C01818=1070.032,30.785,434.123,172.808,24.822,154.487
C01819=1070.038,31.068,434.106,172.809,24.824,154.487
C01820=1070.044,31.317,434.090,172.810,24.827,154.487
C01821=1070.049,31.567,434.074,172.812,24.830,154.488
C01822=1070.056,31.816,434.059,172.813,24.833,154.488
C01823=1070.062,32.066,434.043,172.814,24.835,154.488
C01824=1070.068,32.315,434.027,172.816,24.838,154.489
C01825=1070.073,32.564,434.012,172.817,24.840,154.489
C01826=1070.079,32.814,433.996,172.818,24.843,154.489
C01827=1070.085,33.064,433.980,172.820,24.845,154.490
C01828=1070.091,33.313,433.964,172.821,24.848,154.490
C01829=1070.097,33.563,433.949,172.822,24.851,154.490
C01830=1070.103,33.812,433.933,172.824,24.854,154.491
C01831=1070.108,34.061,433.918,172.826,24.856,154.491
C01832=1070.115,34.310,433.902,172.827,24.859,154.491
C01833=1070.121,34.560,433.887,172.829,24.862,154.492
C01834=1070.127,34.810,433.870,172.830,24.865,154.492
C01835=1070.132,35.060,433.855,172.831,24.867,154.492
C01836=1070.139,35.309,433.839,172.832,24.870,154.493
C01837=1070.145,35.558,433.823,172.834,24.872,154.493
C01838=1070.150,35.807,433.808,172.835,24.875,154.493
C01839=1070.157,36.056,433.792,172.837,24.877,154.494
C01840=1070.162,36.306,433.777,172.838,24.880,154.494
C01841=1070.168,36.556,433.760,172.839,24.883,154.495
C01842=1070.174,36.805,433.744,172.841,24.885,154.495
C01843=1070.181,37.055,433.729,172.842,24.888,154.495
C01844=1070.187,37.304,433.713,172.843,24.890,154.495
C01845=1070.193,37.553,433.697,172.845,24.893,154.496
C01846=1070.198,37.803,433.681,172.846,24.896,154.496
C01847=1070.205,38.052,433.665,172.847,24.898,154.497
C01848=1070.210,38.301,433.649,172.849,24.901,154.497
C01849=1070.216,38.551,433.634,172.851,24.904,154.497
C01850=1070.222,38.800,433.618,172.852,24.906,154.497
C01851=1070.228,39.050,433.601,172.854,24.909,154.498
C01852=1070.233,39.300,433.586,172.855,24.912,154.498
C01853=1070.239,39.549,433.570,172.856,24.915,154.499
C01854=1070.245,39.798,433.553,172.858,24.917,154.499
C01855=1070.251,40.048,433.538,172.859,24.920,154.499
C01856=1070.256,40.297,433.522,172.860,24.923,154.500
C01857=1070.262,40.546,433.506,172.862,24.925,154.500
C01858=1070.268,40.796,433.489,172.863,24.928,154.500
C01859=1070.275,41.045,433.474,172.864,24.930,154.501
C01860=1070.281,41.295,433.458,172.866,24.933,154.501
C01861=1070.286,41.544,433.442,172.867,24.936,154.501
C01862=1070.292,41.793,433.426,172.868,24.939,154.502
C01863=1070.298,42.043,433.409,172.870,24.941,154.502
C01864=1070.304,42.293,433.394,172.871,24.944,154.502
C01865=1070.310,42.542,433.378,172.872,24.946,154.503
C01866=1070.316,42.791,433.361,172.875,24.949,154.503
C01867=1070.322,43.041,433.345,172.876,24.952,154.503
C01868=1070.328,43.290,433.329,172.877,24.955,154.504
C01869=1070.333,43.540,433.313,172.879,24.957,154.504
C01870=1070.339,43.789,433.297,172.880,24.960,154.504
C01871=1070.345,44.038,433.281,172.881,24.963,154.505
C01872=1070.351,44.287,433.265,172.883,24.965,154.505
C01873=1070.357,44.537,433.249,172.884,24.968,154.505
C01874=1070.363,44.786,433.232,172.885,24.970,154.506
C01875=1070.368,45.036,433.216,172.887,24.973,154.506
C01876=1070.374,45.285,433.199,172.888,24.976,154.507
C01877=1070.380,45.534,433.183,172.889,24.979,154.507
C01878=1070.385,45.784,433.168,172.891,24.981,154.507
C01879=1070.391,46.034,433.151,172.892,24.984,154.508
C01880=1070.398,46.316,433.132,172.894,24.988,154.508
C01881=1070.405,46.599,433.114,172.895,24.990,154.508
C01882=1070.411,46.882,433.096,172.897,24.993,154.509
C01883=1070.417,47.164,433.077,172.899,24.997,154.509
C01884=1070.423,47.413,433.061,172.900,25.000,154.510
C01885=1070.429,47.662,433.044,172.901,25.002,154.510
C01886=1070.435,47.912,433.028,172.903,25.005,154.510
C01887=1070.440,48.161,433.011,172.904,25.007,154.511
C01888=1070.446,48.411,432.995,172.905,25.010,154.511
C01889=1070.452,48.660,432.979,172.907,25.013,154.511
C01890=1070.458,48.909,432.963,172.908,25.015,154.512
C01891=1070.464,49.159,432.946,172.909,25.018,154.512
C01892=1070.469,49.408,432.929,172.911,25.021,154.512
C01893=1070.475,49.658,432.913,172.912,25.023,154.513
C01894=1070.481,49.907,432.897,172.913,25.026,154.513
C01895=1070.487,50.156,432.881,172.915,25.029,154.513
C01896=1070.493,50.406,432.864,172.917,25.032,154.514
C01897=1070.498,50.655,432.848,172.918,25.034,154.514
C01898=1070.504,50.905,432.831,172.920,25.037,154.514
C01899=1070.510,51.154,432.815,172.921,25.040,154.515
C01900=1070.517,51.404,432.798,172.922,25.042,154.515
C01901=1070.523,51.654,432.782,172.924,25.045,154.516
C01902=1070.528,51.903,432.765,172.925,25.048,154.516
C01903=1070.534,52.152,432.748,172.926,25.051,154.516
C01904=1070.540,52.401,432.732,172.928,25.053,154.517
C01905=1070.546,52.651,432.716,172.929,25.056,154.517
C01906=1070.551,52.900,432.699,172.930,25.059,154.517
C01907=1070.557,53.150,432.683,172.932,25.061,154.518
C01908=1070.563,53.399,432.666,172.933,25.064,154.518
C01909=1070.569,53.648,432.650,172.934,25.066,154.518
C01910=1070.575,53.897,432.633,172.937,25.069,154.519
C01911=1070.580,54.147,432.616,172.938,25.072,154.519
C01912=1070.586,54.396,432.600,172.939,25.075,154.519
C01913=1070.592,54.645,432.584,172.941,25.078,154.520
C01914=1070.598,54.896,432.567,172.942,25.080,154.520
C01915=1070.604,55.145,432.550,172.943,25.083,154.520
C01916=1070.610,55.394,432.533,172.945,25.085,154.521
C01917=1070.616,55.643,432.517,172.946,25.088,154.521
C01918=1070.622,55.893,432.500,172.948,25.090,154.521
C01919=1070.628,56.142,432.484,172.949,25.093,154.522
C01920=1070.634,56.391,432.467,172.950,25.096,154.522
C01921=1070.640,56.640,432.451,172.951,25.099,154.522
C01922=1070.646,56.891,432.434,172.953,25.101,154.523
C01923=1070.652,57.139,432.417,172.955,25.104,154.523
C01924=1070.658,57.389,432.400,172.956,25.107,154.524
C01925=1070.663,57.638,432.384,172.958,25.109,154.524
C01926=1070.669,57.888,432.367,172.959,25.112,154.524
C01927=1070.675,58.137,432.350,172.961,25.115,154.524
C01928=1070.682,58.387,432.334,172.962,25.117,154.525
C01929=1070.687,58.636,432.317,172.963,25.120,154.525
C01930=1070.693,58.885,432.300,172.965,25.123,154.526
C01931=1070.699,59.134,432.284,172.966,25.125,154.526
C01932=1070.704,59.384,432.267,172.967,25.128,154.526
C01933=1070.711,59.633,432.249,172.969,25.130,154.527
C01934=1070.717,59.883,432.233,172.970,25.133,154.527
C01935=1070.722,60.132,432.216,172.971,25.136,154.527
C01936=1070.729,60.381,432.199,172.974,25.139,154.528
C01937=1070.735,60.630,432.183,172.975,25.141,154.528
C01938=1070.741,60.880,432.165,172.976,25.144,154.528
C01939=1070.747,61.130,432.149,172.978,25.146,154.529
C01940=1070.753,61.379,432.133,172.979,25.149,154.529
C01941=1070.758,61.628,432.115,172.980,25.152,154.529
C01942=1070.765,61.878,432.098,172.982,25.154,154.530
C01943=1070.771,62.127,432.081,172.983,25.157,154.530
C01944=1070.777,62.410,432.063,172.985,25.160,154.530
C01945=1070.784,62.691,432.043,172.987,25.163,154.531
C01946=1070.791,62.974,432.024,172.988,25.166,154.531
C01947=1070.798,63.256,432.005,172.990,25.169,154.531
C01948=1070.803,63.506,431.989,172.992,25.172,154.532
C01949=1070.810,63.755,431.971,172.993,25.174,154.532
C01950=1070.816,64.005,431.955,172.994,25.177,154.532
C01951=1070.821,64.254,431.937,172.996,25.179,154.533
C01952=1070.828,64.504,431.921,172.997,25.182,154.533
C01953=1070.834,64.753,431.903,172.998,25.185,154.534
C01954=1070.839,65.002,431.887,173.000,25.188,154.534
C01955=1070.845,65.251,431.869,173.001,25.190,154.534
C01956=1070.851,65.502,431.852,173.002,25.193,154.535
C01957=1070.857,65.750,431.835,173.005,25.195,154.535
C01958=1070.863,65.999,431.818,173.006,25.198,154.535
C01959=1070.869,66.249,431.801,173.007,25.201,154.536
C01960=1070.875,66.498,431.783,173.009,25.204,154.536
C01961=1070.881,66.748,431.767,173.010,25.206,154.536
C01962=1070.886,66.997,431.750,173.012,25.209,154.537
C01963=1070.892,67.246,431.732,173.013,25.212,154.537
C01964=1070.898,67.496,431.715,173.014,25.214,154.537
C01965=1070.904,67.745,431.698,173.016,25.217,154.538
C01966=1070.910,67.994,431.682,173.017,25.220,154.538
C01967=1070.915,68.243,431.664,173.019,25.222,154.538
C01968=1070.921,68.493,431.646,173.020,25.225,154.539
C01969=1070.927,68.742,431.630,173.022,25.228,154.539
C01970=1070.933,68.991,431.612,173.023,25.230,154.539
C01971=1070.939,69.241,431.594,173.025,25.233,154.540
C01972=1070.945,69.491,431.578,173.026,25.236,154.540
C01973=1070.950,69.740,431.560,173.027,25.239,154.541
C01974=1070.957,69.988,431.543,173.029,25.241,154.541
C01975=1070.962,70.239,431.526,173.030,25.244,154.541
C01976=1070.968,70.488,431.509,173.031,25.246,154.542
C01977=1070.973,70.737,431.491,173.034,25.249,154.542
C01978=1070.980,70.986,431.474,173.035,25.252,154.542
C01979=1070.986,71.236,431.457,173.036,25.255,154.543
C01980=1070.991,71.485,431.439,173.038,25.257,154.543
C01981=1070.997,71.735,431.421,173.039,25.260,154.543
C01982=1071.003,71.983,431.404,173.040,25.263,154.544
C01983=1071.009,72.233,431.388,173.042,25.265,154.544
C01984=1071.015,72.483,431.370,173.043,25.268,154.544
C01985=1071.020,72.732,431.352,173.044,25.271,154.545
C01986=1071.027,72.981,431.335,173.046,25.273,154.545
C01987=1071.032,73.230,431.318,173.048,25.276,154.545
C01988=1071.038,73.480,431.300,173.050,25.279,154.546
C01989=1071.043,73.729,431.283,173.051,25.281,154.546
C01990=1071.049,73.978,431.265,173.052,25.284,154.547
C01991=1071.056,74.227,431.248,173.054,25.287,154.547
C01992=1071.061,74.476,431.230,173.055,25.290,154.547
C01993=1071.067,74.726,431.212,173.056,25.292,154.548
C01994=1071.073,74.976,431.196,173.058,25.295,154.548
C01995=1071.078,75.225,431.178,173.059,25.298,154.548
C01996=1071.085,75.474,431.161,173.061,25.300,154.549
C01997=1071.091,75.723,431.143,173.063,25.303,154.549
C01998=1071.096,75.972,431.126,173.064,25.306,154.549
C01999=1071.102,76.222,431.108,173.065,25.308,154.550
C02000=1071.108,76.471,431.090,173.067,25.311,154.550
C02001=1071.115,76.721,431.073,173.068,25.314,154.550
C02002=1071.120,76.970,431.055,173.070,25.316,154.551
C02003=1071.126,77.219,431.038,173.071,25.319,154.551
C02004=1071.131,77.469,431.020,173.072,25.322,154.551
C02005=1071.137,77.718,431.003,173.075,25.324,154.552
C02006=1071.143,77.968,430.985,173.076,25.327,154.552
C02007=1071.149,78.217,430.967,173.077,25.330,154.552
C02008=1071.155,78.499,430.947,173.079,25.332,154.553
C02009=1071.162,78.781,430.927,173.081,25.336,154.553
C02010=1071.169,79.064,430.907,173.082,25.338,154.554
C02011=1071.176,79.346,430.887,173.083,25.342,154.554
C02012=1071.181,79.595,430.870,173.086,25.345,154.554
C02013=1071.187,79.845,430.852,173.087,25.347,154.555
C02014=1071.193,80.094,430.834,173.088,25.350,154.555
C02015=1071.197,80.343,430.816,173.090,25.353,154.555
C02016=1071.204,80.593,430.798,173.091,25.356,154.556
C02017=1071.209,80.842,430.781,173.092,25.358,154.556
C02018=1071.215,81.092,430.763,173.094,25.361,154.557
C02019=1071.221,81.341,430.745,173.095,25.364,154.557
C02020=1071.227,81.590,430.727,173.097,25.366,154.557
C02021=1071.233,81.839,430.709,173.099,25.369,154.558
C02022=1071.238,82.088,430.691,173.100,25.371,154.558
C02023=1071.244,82.338,430.673,173.102,25.374,154.558
C02024=1071.250,82.587,430.656,173.103,25.377,154.559
C02025=1071.256,82.836,430.638,173.104,25.380,154.559
C02026=1071.261,83.085,430.620,173.106,25.382,154.559
C02027=1071.268,83.335,430.602,173.107,25.385,154.560
C02028=1071.273,83.584,430.584,173.109,25.388,154.560
C02029=1071.280,83.833,430.566,173.111,25.391,154.560
C02030=1071.285,84.082,430.549,173.112,25.393,154.561
C02031=1071.291,84.331,430.531,173.113,25.396,154.561
C02032=1071.296,84.581,430.513,173.115,25.398,154.561
C02033=1071.301,84.830,430.495,173.116,25.401,154.562
C02034=1071.308,85.080,430.476,173.117,25.404,154.562
C02035=1071.313,85.329,430.459,173.120,25.407,154.562
C02036=1071.320,85.578,430.441,173.121,25.410,154.563
C02037=1071.325,85.827,430.423,173.123,25.412,154.563
C02038=1071.331,86.077,430.405,173.124,25.415,154.564
C02039=1071.337,86.326,430.387,173.125,25.417,154.564
C02040=1071.343,86.575,430.369,173.127,25.420,154.564
C02041=1071.349,86.825,430.351,173.128,25.423,154.565
C02042=1071.355,87.073,430.333,173.129,25.425,154.565
C02043=1071.360,87.324,430.314,173.132,25.428,154.565
C02044=1071.366,87.573,430.297,173.133,25.431,154.566
C02045=1071.372,87.822,430.279,173.134,25.433,154.566
C02046=1071.378,88.071,430.261,173.136,25.436,154.566
C02047=1071.384,88.320,430.243,173.137,25.439,154.567
C02048=1071.390,88.570,430.225,173.139,25.441,154.567
C02049=1071.396,88.819,430.207,173.141,25.444,154.567
C02050=1071.402,89.068,430.189,173.142,25.447,154.568
C02051=1071.407,89.318,430.170,173.144,25.449,154.568
C02052=1071.413,89.567,430.152,173.145,25.452,154.568
C02053=1071.419,89.816,430.134,173.146,25.455,154.569
C02054=1071.425,90.066,430.116,173.148,25.457,154.569
C02055=1071.431,90.314,430.098,173.149,25.460,154.569
C02056=1071.437,90.564,430.080,173.152,25.462,154.570
C02057=1071.443,90.813,430.061,173.153,25.465,154.570
C02058=1071.448,91.062,430.043,173.154,25.468,154.570
C02059=1071.454,91.312,430.025,173.156,25.470,154.571
C02060=1071.460,91.560,430.007,173.157,25.473,154.571
C02061=1071.465,91.810,429.988,173.158,25.476,154.571
C02062=1071.471,92.059,429.970,173.160,25.478,154.572
C02063=1071.477,92.309,429.952,173.162,25.482,154.572
C02064=1071.482,92.557,429.933,173.163,25.484,154.573
C02065=1071.489,92.807,429.915,173.165,25.487,154.573
C02066=1071.494,93.057,429.897,173.166,25.489,154.573
C02067=1071.500,93.306,429.879,173.167,25.492,154.574
C02068=1071.506,93.555,429.861,173.169,25.495,154.574
C02069=1071.511,93.804,429.842,173.171,25.498,154.574
C02070=1071.517,94.054,429.824,173.173,25.500,154.575
C02071=1071.524,94.303,429.805,173.174,25.503,154.575
C02072=1071.530,94.585,429.784,173.175,25.506,154.575
C02073=1071.536,94.868,429.764,173.178,25.509,154.576
C02074=1071.542,95.150,429.743,173.179,25.512,154.576
C02075=1071.550,95.432,429.722,173.181,25.515,154.577
C02076=1071.555,95.681,429.703,173.182,25.518,154.577
C02077=1071.561,95.931,429.685,173.184,25.521,154.577
C02078=1071.566,96.180,429.666,173.185,25.523,154.578
C02079=1071.572,96.429,429.648,173.187,25.526,154.578
C02080=1071.578,96.678,429.630,173.189,25.528,154.578
C02081=1071.583,96.928,429.611,173.190,25.531,154.579
C02082=1071.590,97.177,429.593,173.192,25.534,154.579
C02083=1071.595,97.426,429.574,173.193,25.536,154.579
C02084=1071.601,97.675,429.556,173.194,25.539,154.580
C02085=1071.607,97.924,429.537,173.196,25.542,154.580
C02086=1071.613,98.174,429.518,173.198,25.545,154.580
C02087=1071.618,98.423,429.501,173.200,25.547,154.581
C02088=1071.624,98.672,429.481,173.201,25.550,154.581
C02089=1071.631,98.921,429.463,173.202,25.552,154.581
C02090=1071.636,99.172,429.444,173.204,25.555,154.582
C02091=1071.642,99.420,429.426,173.205,25.557,154.582
C02092=1071.648,99.669,429.407,173.207,25.561,154.582
C02093=1071.654,99.919,429.389,173.209,25.563,154.583
C02094=1071.659,100.168,429.370,173.210,25.566,154.583
C02095=1071.665,100.417,429.351,173.212,25.568,154.583
C02096=1071.671,100.666,429.332,173.213,25.571,154.584
C02097=1071.677,100.916,429.314,173.215,25.574,154.584
C02098=1071.683,101.165,429.296,173.217,25.576,154.585
C02099=1071.688,101.414,429.276,173.218,25.579,154.585
C02100=1071.695,101.663,429.258,173.219,25.582,154.585
C02101=1071.700,101.912,429.240,173.221,25.584,154.586
C02102=1071.705,102.162,429.220,173.223,25.587,154.586
C02103=1071.712,102.411,429.202,173.224,25.590,154.586
C02104=1071.717,102.660,429.183,173.226,25.592,154.587
C02105=1071.722,102.909,429.164,173.227,25.595,154.587
C02106=1071.729,103.159,429.146,173.229,25.597,154.587
C02107=1071.734,103.408,429.127,173.230,25.600,154.588
C02108=1071.739,103.657,429.108,173.232,25.603,154.588
C02109=1071.746,103.906,429.089,173.234,25.606,154.588
C02110=1071.751,104.156,429.070,173.235,25.609,154.589
C02111=1071.757,104.404,429.051,173.237,25.611,154.589
C02112=1071.763,104.654,429.033,173.238,25.614,154.589
C02113=1071.768,104.904,429.014,173.240,25.616,154.590
C02114=1071.774,105.153,428.994,173.242,25.619,154.590
C02115=1071.780,105.401,428.976,173.243,25.622,154.590
C02116=1071.786,105.651,428.957,173.244,25.624,154.591
C02117=1071.791,105.900,428.938,173.246,25.627,154.591
C02118=1071.798,106.149,428.919,173.248,25.630,154.591
C02119=1071.803,106.398,428.900,173.249,25.633,154.592
C02120=1071.808,106.648,428.881,173.251,25.635,154.592
C02121=1071.815,106.897,428.862,173.252,25.638,154.593
C02122=1071.821,107.146,428.843,173.254,25.640,154.593
C02123=1071.826,107.396,428.824,173.256,25.643,154.593
C02124=1071.832,107.644,428.805,173.257,25.646,154.593
C02125=1071.838,107.893,428.786,173.259,25.648,154.594
C02126=1071.843,108.143,428.767,173.260,25.651,154.594
C02127=1071.849,108.392,428.748,173.263,25.654,154.595
C02128=1071.856,108.641,428.729,173.264,25.656,154.595
C02129=1071.861,108.890,428.710,173.265,25.659,154.595
C02130=1071.866,109.140,428.691,173.267,25.661,154.596
C02131=1071.873,109.389,428.672,173.268,25.664,154.596
C02132=1071.878,109.638,428.653,173.271,25.667,154.596
C02133=1071.884,109.888,428.634,173.272,25.670,154.597
C02134=1071.890,110.137,428.615,173.273,25.672,154.597
C02135=1071.896,110.385,428.596,173.275,25.675,154.597
C02136=1071.902,110.668,428.574,173.277,25.678,154.598
C02137=1071.909,110.950,428.552,173.278,25.681,154.598
C02138=1071.915,111.233,428.531,173.281,25.684,154.598
C02139=1071.922,111.516,428.509,173.282,25.687,154.599
C02140=1071.928,111.765,428.490,173.284,25.690,154.599
C02141=1071.933,112.014,428.471,173.286,25.692,154.599
C02142=1071.939,112.263,428.451,173.287,25.695,154.600
C02143=1071.944,112.512,428.432,173.288,25.698,154.600
C02144=1071.951,112.761,428.413,173.290,25.700,154.600
C02145=1071.957,113.011,428.394,173.292,25.703,154.601
C02146=1071.962,113.260,428.375,173.294,25.705,154.601
C02147=1071.968,113.509,428.356,173.295,25.708,154.602
C02148=1071.974,113.758,428.336,173.296,25.710,154.602
C02149=1071.980,114.008,428.317,173.299,25.714,154.602
C02150=1071.985,114.256,428.298,173.300,25.716,154.602
C02151=1071.990,114.506,428.278,173.302,25.719,154.603
C02152=1071.996,114.755,428.259,173.303,25.722,154.603
C02153=1072.002,115.004,428.239,173.305,25.724,154.604
C02154=1072.008,115.254,428.220,173.307,25.727,154.604
C02155=1072.013,115.503,428.201,173.308,25.729,154.604
C02156=1072.019,115.751,428.181,173.309,25.732,154.605
C02157=1072.025,116.000,428.162,173.312,25.735,154.605
C02158=1072.030,116.250,428.143,173.313,25.738,154.605
C02159=1072.036,116.499,428.123,173.314,25.741,154.606
C02160=1072.042,116.748,428.103,173.316,25.743,154.606
C02161=1072.047,116.998,428.084,173.317,25.746,154.606
C02162=1072.053,117.247,428.064,173.320,25.749,154.607
C02163=1072.058,117.495,428.045,173.321,25.751,154.607
C02164=1072.064,117.745,428.026,173.322,25.754,154.608
C02165=1072.069,117.994,428.006,173.324,25.756,154.608
C02166=1072.075,118.243,427.986,173.326,25.759,154.608
C02167=1072.081,118.493,427.967,173.328,25.762,154.608
C02168=1072.087,118.742,427.948,173.329,25.765,154.609
C02169=1072.093,118.991,427.928,173.330,25.767,154.609
C02170=1072.098,119.240,427.909,173.333,25.770,154.610
C02171=1072.104,119.489,427.888,173.334,25.773,154.610
C02172=1072.109,119.739,427.869,173.336,25.775,154.610
C02173=1072.115,119.988,427.850,173.338,25.778,154.611
C02174=1072.121,120.237,427.830,173.339,25.781,154.611
C02175=1072.126,120.486,427.811,173.341,25.783,154.611
C02176=1072.132,120.735,427.791,173.342,25.786,154.612
C02177=1072.138,120.984,427.772,173.344,25.789,154.612
C02178=1072.143,121.233,427.751,173.346,25.791,154.612
C02179=1072.149,121.483,427.732,173.347,25.794,154.613
C02180=1072.155,121.731,427.712,173.349,25.796,154.613
C02181=1072.160,121.981,427.693,173.351,25.799,154.613
C02182=1072.166,122.230,427.673,173.352,25.802,154.614
C02183=1072.172,122.479,427.653,173.354,25.805,154.614
C02184=1072.178,122.728,427.633,173.355,25.807,154.614
C02185=1072.183,122.978,427.614,173.358,25.810,154.615
C02186=1072.189,123.226,427.594,173.359,25.812,154.615
C02187=1072.195,123.476,427.574,173.360,25.815,154.615
C02188=1072.201,123.725,427.554,173.363,25.818,154.616
C02189=1072.206,123.974,427.535,173.364,25.821,154.616
C02190=1072.212,124.223,427.515,173.366,25.823,154.616
C02191=1072.217,124.473,427.495,173.367,25.826,154.617
C02192=1072.223,124.721,427.475,173.369,25.828,154.617
C02193=1072.229,124.970,427.455,173.371,25.831,154.617
C02194=1072.235,125.220,427.436,173.372,25.833,154.618
C02195=1072.241,125.469,427.416,173.374,25.837,154.618
C02196=1072.246,125.718,427.396,173.376,25.839,154.618
C02197=1072.253,125.968,427.376,173.377,25.842,154.619
C02198=1072.259,126.217,427.356,173.379,25.844,154.619
C02199=1072.264,126.466,427.337,173.381,25.847,154.619
C02200=1072.270,126.748,427.314,173.382,25.850,154.620
C02201=1072.277,127.031,427.292,173.385,25.853,154.620
C02202=1072.284,127.313,427.269,173.387,25.856,154.620
C02203=1072.290,127.595,427.247,173.388,25.859,154.621
C02204=1072.296,127.844,427.227,173.390,25.861,154.621
C02205=1072.301,128.093,427.206,173.392,25.864,154.621
C02206=1072.308,128.343,427.187,173.394,25.866,154.622
C02207=1072.314,128.592,427.167,173.395,25.869,154.622
C02208=1072.319,128.841,427.147,173.397,25.872,154.622
C02209=1072.325,129.090,427.126,173.399,25.875,154.623
C02210=1072.330,129.339,427.107,173.400,25.877,154.623
C02211=1072.336,129.588,427.087,173.403,25.880,154.624
C02212=1072.342,129.837,427.067,173.404,25.882,154.624
C02213=1072.348,130.086,427.046,173.406,25.885,154.624
C02214=1072.354,130.336,427.027,173.407,25.887,154.625
C02215=1072.360,130.585,427.007,173.409,25.890,154.625
C02216=1072.366,130.834,426.987,173.411,25.893,154.625
C02217=1072.371,131.083,426.966,173.412,25.895,154.625
C02218=1072.377,131.332,426.946,173.415,25.898,154.626
C02219=1072.383,131.580,426.926,173.416,25.901,154.626
C02220=1072.389,131.831,426.907,173.417,25.903,154.626
C02221=1072.395,132.080,426.886,173.420,25.906,154.627
C02222=1072.401,132.329,426.866,173.421,25.908,154.627
C02223=1072.406,132.578,426.846,173.423,25.911,154.627
C02224=1072.412,132.827,426.826,173.425,25.914,154.628
C02225=1072.417,133.076,426.805,173.426,25.917,154.628
C02226=1072.423,133.324,426.785,173.428,25.919,154.628
C02227=1072.429,133.574,426.764,173.430,25.922,154.629
C02228=1072.435,133.823,426.744,173.432,25.924,154.629
C02229=1072.440,134.073,426.725,173.433,25.927,154.629
C02230=1072.446,134.322,426.705,173.435,25.930,154.630
C02231=1072.451,134.571,426.684,173.437,25.932,154.630
C02232=1072.457,134.820,426.664,173.438,25.935,154.630
C02233=1072.463,135.069,426.644,173.441,25.937,154.631
C02234=1072.469,135.318,426.623,173.442,25.940,154.631
C02235=1072.474,135.567,426.603,173.443,25.943,154.631
C02236=1072.480,135.816,426.583,173.446,25.946,154.632
C02237=1072.486,136.065,426.562,173.447,25.948,154.632
C02238=1072.492,136.314,426.542,173.449,25.951,154.632
C02239=1072.497,136.564,426.521,173.451,25.953,154.633
C02240=1072.503,136.813,426.501,173.452,25.956,154.633
C02241=1072.509,137.062,426.481,173.454,25.959,154.633
C02242=1072.514,137.311,426.460,173.456,25.962,154.634
C02243=1072.520,137.560,426.440,173.458,25.964,154.634
C02244=1072.526,137.809,426.419,173.459,25.966,154.634
C02245=1072.532,138.058,426.399,173.461,25.969,154.635
C02246=1072.537,138.307,426.378,173.463,25.972,154.635
C02247=1072.543,138.556,426.358,173.464,25.974,154.635
C02248=1072.549,138.805,426.338,173.467,25.977,154.636
C02249=1072.555,139.055,426.317,173.468,25.980,154.636
C02250=1072.561,139.304,426.297,173.471,25.982,154.636
C02251=1072.566,139.553,426.276,173.472,25.985,154.637
C02252=1072.571,139.802,426.256,173.473,25.988,154.637
C02253=1072.578,140.051,426.235,173.476,25.990,154.637
C02254=1072.583,140.300,426.214,173.477,25.993,154.638
C02255=1072.589,140.549,426.194,173.479,25.995,154.638
C02256=1072.594,140.798,426.174,173.481,25.998,154.638
C02257=1072.600,141.048,426.153,173.482,26.001,154.639
C02258=1072.606,141.296,426.131,173.484,26.004,154.639
C02259=1072.612,141.545,426.111,173.486,26.006,154.639
C02260=1072.617,141.794,426.091,173.488,26.009,154.640
C02261=1072.623,142.044,426.070,173.490,26.012,154.640
C02262=1072.628,142.293,426.049,173.491,26.014,154.640
C02263=1072.635,142.541,426.029,173.493,26.017,154.641
C02264=1072.640,142.824,426.005,173.495,26.020,154.641
C02265=1072.647,143.106,425.982,173.497,26.023,154.641
C02266=1072.654,143.388,425.958,173.499,26.026,154.642
C02267=1072.659,143.670,425.935,173.501,26.029,154.642
C02268=1072.665,143.920,425.913,173.503,26.032,154.643
C02269=1072.671,144.168,425.893,173.505,26.034,154.643
C02270=1072.677,144.418,425.873,173.506,26.037,154.643
C02271=1072.683,144.667,425.851,173.509,26.040,154.644
C02272=1072.688,144.916,425.831,173.510,26.042,154.644
C02273=1072.694,145.165,425.811,173.512,26.045,154.644
C02274=1072.700,145.414,425.789,173.514,26.047,154.645
C02275=1072.706,145.663,425.769,173.515,26.050,154.645
C02276=1072.711,145.912,425.747,173.518,26.053,154.645
C02277=1072.717,146.161,425.726,173.519,26.056,154.646
C02278=1072.723,146.410,425.706,173.521,26.058,154.646
C02279=1072.728,146.659,425.685,173.523,26.060,154.646
C02280=1072.734,146.909,425.664,173.524,26.063,154.647
C02281=1072.740,147.157,425.643,173.527,26.066,154.647
C02282=1072.745,147.406,425.622,173.528,26.069,154.647
C02283=1072.751,147.656,425.601,173.530,26.071,154.648
C02284=1072.757,147.904,425.581,173.532,26.074,154.648
C02285=1072.763,148.154,425.560,173.534,26.076,154.648
C02286=1072.769,148.403,425.539,173.536,26.079,154.648
C02287=1072.774,148.652,425.518,173.537,26.082,154.649
C02288=1072.780,148.901,425.496,173.540,26.084,154.649
C02289=1072.785,149.150,425.476,173.541,26.087,154.650
C02290=1072.791,149.398,425.455,173.543,26.089,154.650
C02291=1072.797,149.648,425.434,173.545,26.093,154.650
C02292=1072.802,149.897,425.412,173.546,26.095,154.651
C02293=1072.808,150.146,425.392,173.549,26.098,154.651
C02294=1072.814,150.395,425.370,173.550,26.100,154.651
C02295=1072.819,150.644,425.349,173.552,26.103,154.652
C02296=1072.825,150.893,425.328,173.554,26.106,154.652
C02297=1072.831,151.142,425.307,173.555,26.108,154.652
C02298=1072.836,151.391,425.286,173.558,26.111,154.653
C02299=1072.842,151.640,425.265,173.559,26.114,154.653
C02300=1072.847,151.889,425.244,173.562,26.116,154.653
C02301=1072.854,152.139,425.222,173.563,26.119,154.653
C02302=1072.859,152.387,425.201,173.565,26.121,154.654
C02303=1072.864,152.636,425.181,173.567,26.124,154.654
C02304=1072.871,152.885,425.159,173.568,26.127,154.655
C02305=1072.876,153.134,425.138,173.571,26.129,154.655
C02306=1072.882,153.384,425.117,173.572,26.132,154.655
C02307=1072.888,153.632,425.095,173.575,26.135,154.655
C02308=1072.894,153.882,425.074,173.576,26.138,154.656
C02309=1072.899,154.131,425.053,173.578,26.140,154.656
C02310=1072.904,154.380,425.031,173.580,26.143,154.657
C02311=1072.910,154.629,425.010,173.581,26.145,154.657
C02312=1072.916,154.877,424.988,173.584,26.148,154.657
C02313=1072.921,155.127,424.968,173.585,26.151,154.658
C02314=1072.927,155.375,424.946,173.588,26.153,154.658
C02315=1072.933,155.625,424.925,173.589,26.156,154.658
C02316=1072.939,155.873,424.903,173.591,26.159,154.658
C02317=1072.945,156.123,424.882,173.593,26.161,154.659
C02318=1072.949,156.372,424.861,173.595,26.164,154.659
C02319=1072.956,156.621,424.839,173.597,26.167,154.660
C02320=1072.961,156.870,424.818,173.599,26.169,154.660
C02321=1072.967,157.119,424.796,173.600,26.172,154.660
C02322=1072.973,157.368,424.776,173.603,26.175,154.660
C02323=1072.978,157.617,424.753,173.604,26.178,154.661
C02324=1072.984,157.866,424.732,173.606,26.180,154.661
C02325=1072.990,158.115,424.710,173.608,26.182,154.661
C02326=1072.995,158.364,424.689,173.610,26.185,154.662
C02327=1073.001,158.613,424.667,173.612,26.188,154.662
C02328=1073.007,158.895,424.643,173.614,26.191,154.662
C02329=1073.014,159.177,424.618,173.617,26.194,154.663
C02330=1073.020,159.459,424.594,173.618,26.197,154.663
C02331=1073.027,159.741,424.570,173.620,26.200,154.664
C02332=1073.032,159.989,424.548,173.623,26.203,154.664
C02333=1073.038,160.239,424.526,173.624,26.205,154.664
C02334=1073.044,160.487,424.505,173.627,26.208,154.665
C02335=1073.050,160.737,424.484,173.628,26.211,154.665
C02336=1073.054,160.986,424.462,173.630,26.213,154.665
C02337=1073.061,161.235,424.441,173.632,26.216,154.666
C02338=1073.067,161.484,424.419,173.634,26.219,154.666
C02339=1073.072,161.733,424.397,173.636,26.221,154.666
C02340=1073.078,161.982,424.376,173.638,26.224,154.667
C02341=1073.083,162.231,424.354,173.639,26.227,154.667
C02342=1073.089,162.480,424.331,173.642,26.229,154.667
C02343=1073.094,162.728,424.310,173.643,26.232,154.668
C02344=1073.100,162.978,424.288,173.646,26.235,154.668
C02345=1073.105,163.226,424.266,173.647,26.238,154.668
C02346=1073.110,163.476,424.244,173.649,26.241,154.669
C02347=1073.116,163.725,424.223,173.651,26.243,154.669
C02348=1073.121,163.974,424.200,173.653,26.246,154.669
C02349=1073.127,164.223,424.179,173.655,26.249,154.670
C02350=1073.132,164.472,424.157,173.657,26.251,154.670
C02351=1073.138,164.721,424.136,173.659,26.254,154.670
C02352=1073.143,164.970,424.113,173.661,26.257,154.671
C02353=1073.149,165.218,424.091,173.662,26.260,154.671
C02354=1073.155,165.467,424.069,173.665,26.263,154.672
C02355=1073.159,165.716,424.047,173.666,26.265,154.672
C02356=1073.166,165.965,424.026,173.668,26.268,154.672
C02357=1073.171,166.215,424.003,173.670,26.270,154.672
C02358=1073.177,166.463,423.981,173.672,26.273,154.673
C02359=1073.182,166.712,423.959,173.674,26.276,154.673
C02360=1073.187,166.961,423.937,173.676,26.279,154.674
C02361=1073.193,167.210,423.916,173.678,26.281,154.674
C02362=1073.199,167.460,423.893,173.680,26.284,154.674
C02363=1073.205,167.708,423.871,173.681,26.287,154.675
C02364=1073.210,167.957,423.849,173.684,26.290,154.675
C02365=1073.215,168.206,423.827,173.686,26.293,154.675
C02366=1073.221,168.455,423.805,173.688,26.295,154.676
C02367=1073.227,168.704,423.783,173.690,26.298,154.676
C02368=1073.232,168.953,423.762,173.692,26.300,154.676
C02369=1073.238,169.202,423.739,173.694,26.303,154.677
C02370=1073.243,169.451,423.716,173.695,26.306,154.677
C02371=1073.249,169.700,423.695,173.698,26.309,154.677
C02372=1073.254,169.949,423.673,173.699,26.311,154.678
C02373=1073.260,170.198,423.650,173.702,26.314,154.678
C02374=1073.266,170.447,423.629,173.704,26.317,154.678
C02375=1073.271,170.696,423.606,173.705,26.319,154.679
C02376=1073.278,170.945,423.584,173.708,26.322,154.679
C02377=1073.282,171.194,423.562,173.709,26.325,154.679
C02378=1073.288,171.442,423.539,173.712,26.328,154.680
C02379=1073.294,171.692,423.518,173.713,26.330,154.680
C02380=1073.299,171.940,423.496,173.715,26.333,154.680
C02381=1073.305,172.189,423.473,173.717,26.336,154.681
C02382=1073.311,172.439,423.451,173.719,26.339,154.681
C02383=1073.317,172.687,423.428,173.722,26.341,154.681
C02384=1073.322,172.936,423.406,173.723,26.344,154.682
C02385=1073.328,173.185,423.384,173.726,26.347,154.682
C02386=1073.333,173.434,423.362,173.727,26.349,154.682
C02387=1073.339,173.683,423.339,173.729,26.352,154.683
C02388=1073.345,173.932,423.318,173.732,26.355,154.683
C02389=1073.350,174.181,423.295,173.733,26.357,154.683
C02390=1073.356,174.430,423.272,173.736,26.360,154.684
C02391=1073.362,174.679,423.249,173.737,26.363,154.684
C02392=1073.368,174.960,423.225,173.739,26.366,154.684
C02393=1073.375,175.242,423.199,173.742,26.369,154.685
C02394=1073.381,175.523,423.174,173.744,26.372,154.685
C02395=1073.388,175.805,423.149,173.746,26.375,154.686
C02396=1073.393,176.054,423.126,173.749,26.378,154.686
C02397=1073.399,176.302,423.104,173.750,26.380,154.686
C02398=1073.404,176.552,423.081,173.753,26.383,154.686
C02399=1073.410,176.801,423.059,173.755,26.386,154.687
C02400=1073.416,177.050,423.037,173.757,26.388,154.687
C02401=1073.422,177.299,423.014,173.759,26.391,154.687
C02402=1073.428,177.548,422.992,173.760,26.394,154.688
C02403=1073.433,177.796,422.970,173.763,26.396,154.688
C02404=1073.439,178.045,422.947,173.765,26.399,154.688
C02405=1073.444,178.294,422.924,173.767,26.401,154.689
C02406=1073.451,178.543,422.902,173.769,26.405,154.689
C02407=1073.456,178.792,422.879,173.771,26.407,154.689
C02408=1073.462,179.041,422.856,173.773,26.410,154.690
C02409=1073.467,179.291,422.834,173.775,26.412,154.690
C02410=1073.474,179.539,422.812,173.777,26.415,154.690
C02411=1073.479,179.787,422.789,173.779,26.418,154.691
C02412=1073.485,180.036,422.766,173.782,26.420,154.691
C02413=1073.490,180.286,422.744,173.783,26.423,154.691
C02414=1073.496,180.535,422.721,173.786,26.426,154.692
C02415=1073.502,180.783,422.699,173.788,26.429,154.692
C02416=1073.508,181.032,422.676,173.789,26.431,154.692
C02417=1073.514,181.281,422.653,173.792,26.434,154.693
C02418=1073.519,181.531,422.630,173.794,26.437,154.693
C02419=1073.526,181.779,422.608,173.796,26.439,154.693
C02420=1073.531,182.028,422.585,173.798,26.442,154.694
C02421=1073.537,182.277,422.562,173.800,26.444,154.694
C02422=1073.543,182.526,422.539,173.802,26.447,154.694
C02423=1073.549,182.775,422.516,173.804,26.450,154.695
C02424=1073.554,183.024,422.493,173.806,26.452,154.695
C02425=1073.561,183.273,422.472,173.808,26.455,154.695
C02426=1073.566,183.522,422.449,173.811,26.458,154.696
C02427=1073.572,183.771,422.426,173.812,26.461,154.696
C02428=1073.578,184.020,422.403,173.815,26.463,154.696
C02429=1073.583,184.269,422.380,173.817,26.466,154.697
C02430=1073.590,184.517,422.358,173.819,26.468,154.697
C02431=1073.596,184.766,422.335,173.821,26.471,154.697
C02432=1073.601,185.015,422.312,173.823,26.474,154.698
C02433=1073.606,185.263,422.289,173.826,26.477,154.698
C02434=1073.612,185.512,422.266,173.827,26.479,154.698
C02435=1073.617,185.761,422.243,173.830,26.482,154.699
C02436=1073.623,186.010,422.220,173.832,26.486,154.699
C02437=1073.628,186.259,422.196,173.833,26.488,154.699
C02438=1073.634,186.508,422.173,173.836,26.491,154.700
C02439=1073.639,186.757,422.150,173.838,26.494,154.700
C02440=1073.645,187.006,422.127,173.840,26.496,154.700
C02441=1073.650,187.255,422.104,173.842,26.499,154.701
C02442=1073.656,187.504,422.081,173.844,26.502,154.701
C02443=1073.661,187.752,422.058,173.846,26.505,154.701
C02444=1073.667,188.001,422.035,173.848,26.508,154.702
C02445=1073.672,188.250,422.011,173.851,26.511,154.702
C02446=1073.678,188.499,421.988,173.852,26.513,154.702
C02447=1073.683,188.748,421.965,173.854,26.516,154.703
C02448=1073.689,188.996,421.942,173.857,26.519,154.703
C02449=1073.694,189.246,421.919,173.859,26.522,154.703
C02450=1073.700,189.495,421.896,173.861,26.524,154.704
C02451=1073.706,189.743,421.872,173.863,26.527,154.704
C02452=1073.712,189.992,421.849,173.865,26.530,154.705
C02453=1073.717,190.241,421.826,173.867,26.533,154.705
C02454=1073.722,190.490,421.803,173.869,26.535,154.705
C02455=1073.728,190.739,421.780,173.872,26.539,154.706
C02456=1073.735,191.020,421.753,173.874,26.542,154.706
C02457=1073.740,191.301,421.727,173.876,26.545,154.706
C02458=1073.747,191.583,421.700,173.879,26.548,154.707
C02459=1073.754,191.864,421.674,173.881,26.551,154.707
C02460=1073.759,192.113,421.650,173.883,26.554,154.708
C02461=1073.765,192.362,421.627,173.886,26.557,154.708
C02462=1073.771,192.610,421.604,173.887,26.559,154.708
C02463=1073.776,192.859,421.580,173.890,26.562,154.709
C02464=1073.782,193.108,421.557,173.892,26.565,154.709
C02465=1073.788,193.356,421.533,173.895,26.568,154.709
C02466=1073.793,193.606,421.510,173.896,26.571,154.710
C02467=1073.798,193.854,421.487,173.898,26.574,154.710
C02468=1073.804,194.103,421.463,173.901,26.576,154.710
C02469=1073.809,194.352,421.440,173.903,26.579,154.711
C02470=1073.815,194.601,421.417,173.905,26.582,154.711
C02471=1073.821,194.849,421.393,173.907,26.585,154.711
C02472=1073.827,195.099,421.369,173.909,26.588,154.712
C02473=1073.833,195.347,421.346,173.912,26.590,154.712
C02474=1073.838,195.596,421.322,173.913,26.593,154.712
C02475=1073.844,195.845,421.298,173.916,26.596,154.713
C02476=1073.850,196.094,421.275,173.918,26.599,154.713
C02477=1073.855,196.343,421.252,173.920,26.602,154.713
C02478=1073.861,196.591,421.228,173.922,26.604,154.714
C02479=1073.866,196.840,421.205,173.924,26.607,154.714
C02480=1073.872,197.089,421.181,173.927,26.610,154.715
C02481=1073.878,197.338,421.158,173.929,26.613,154.715
C02482=1073.883,197.587,421.133,173.932,26.616,154.715
C02483=1073.889,197.835,421.110,173.933,26.618,154.715
C02484=1073.895,198.084,421.087,173.935,26.621,154.716
C02485=1073.901,198.333,421.062,173.938,26.624,154.716
C02486=1073.907,198.582,421.039,173.940,26.627,154.717
C02487=1073.912,198.831,421.015,173.942,26.629,154.717
C02488=1073.918,199.080,420.992,173.944,26.632,154.717
C02489=1073.924,199.328,420.968,173.947,26.635,154.718
C02490=1073.930,199.577,420.944,173.949,26.638,154.718
C02491=1073.935,199.826,420.921,173.951,26.641,154.718
C02492=1073.941,200.075,420.897,173.954,26.644,154.719
C02493=1073.946,200.324,420.874,173.955,26.646,154.719
C02494=1073.952,200.573,420.849,173.958,26.649,154.719
C02495=1073.958,200.821,420.825,173.960,26.652,154.720
C02496=1073.964,201.070,420.802,173.962,26.655,154.720
C02497=1073.969,201.319,420.778,173.965,26.658,154.720
C02498=1073.976,201.568,420.754,173.966,26.660,154.721
C02499=1073.981,201.816,420.730,173.969,26.663,154.721
C02500=1073.987,202.065,420.707,173.971,26.666,154.721
C02501=1073.992,202.314,420.683,173.974,26.668,154.722
C02502=1073.999,202.563,420.659,173.976,26.672,154.722
C02503=1074.004,202.811,420.634,173.978,26.675,154.722
C02504=1074.009,203.060,420.611,173.980,26.677,154.723
C02505=1074.015,203.309,420.587,173.982,26.680,154.723
C02506=1074.021,203.558,420.563,173.985,26.683,154.724
C02507=1074.026,203.807,420.538,173.987,26.686,154.724
C02508=1074.032,204.055,420.514,173.989,26.689,154.724
C02509=1074.038,204.304,420.491,173.992,26.692,154.725
C02510=1074.043,204.553,420.467,173.993,26.694,154.725
C02511=1074.049,204.802,420.442,173.996,26.697,154.725
C02512=1074.055,205.050,420.419,173.998,26.701,154.726
C02513=1074.060,205.299,420.394,174.000,26.703,154.726
C02514=1074.066,205.548,420.370,174.003,26.706,154.726
C02515=1074.071,205.797,420.345,174.005,26.709,154.727
C02516=1074.077,206.045,420.322,174.007,26.712,154.727
C02517=1074.083,206.295,420.298,174.009,26.715,154.728
C02518=1074.088,206.544,420.274,174.011,26.718,154.728
C02519=1074.094,206.792,420.250,174.014,26.721,154.728
C02520=1074.118,207.831,420.148,174.137,26.785,154.729
C02521=1074.127,208.246,420.107,174.140,26.791,154.730
C02522=1074.137,208.660,420.065,174.144,26.798,154.731
C02523=1074.147,209.075,420.025,174.147,26.804,154.732
C02524=1074.156,209.489,419.982,174.150,26.811,154.733
C02525=1074.162,209.738,419.958,174.153,26.814,154.733
C02526=1074.168,209.986,419.933,174.155,26.818,154.734
C02527=1074.174,210.235,419.907,174.157,26.822,154.735
C02528=1074.180,210.484,419.883,174.159,26.826,154.735
C02529=1074.185,210.732,419.858,174.161,26.830,154.736
C02530=1074.191,210.981,419.833,174.164,26.834,154.736
C02531=1074.197,211.230,419.808,174.165,26.837,154.737
C02532=1074.203,211.478,419.783,174.167,26.841,154.738
C02533=1074.208,211.728,419.758,174.169,26.845,154.738
C02534=1074.214,211.976,419.732,174.172,26.849,154.739
C02535=1074.220,212.224,419.707,174.174,26.852,154.739
C02536=1074.226,212.474,419.683,174.176,26.856,154.740
C02537=1074.232,212.722,419.657,174.178,26.860,154.740
C02538=1074.238,212.970,419.632,174.180,26.864,154.741
C02539=1074.243,213.220,419.607,174.183,26.868,154.741
C02540=1074.249,213.469,419.582,174.185,26.872,154.742
C02541=1074.255,213.717,419.557,174.186,26.875,154.743
C02542=1074.261,213.965,419.532,174.188,26.879,154.743
C02543=1074.266,214.215,419.506,174.191,26.883,154.744
C02544=1074.272,214.463,419.481,174.193,26.887,154.744
C02545=1074.278,214.711,419.456,174.195,26.891,154.745
C02546=1074.283,214.960,419.430,174.197,26.895,154.746
C02547=1074.289,215.208,419.405,174.200,26.898,154.746
C02548=1074.295,215.458,419.381,174.202,26.902,154.747
C02549=1074.300,215.707,419.355,174.204,26.906,154.747
C02550=1074.306,215.955,419.330,174.206,26.910,154.748
C02551=1074.312,216.203,419.304,174.208,26.914,154.749
C02552=1074.318,216.452,419.279,174.211,26.918,154.749
C02553=1074.324,216.701,419.253,174.212,26.921,154.750
C02554=1074.329,216.949,419.228,174.214,26.925,154.750
C02555=1074.336,217.198,419.203,174.217,26.929,154.751
C02556=1074.341,217.447,419.178,174.219,26.933,154.751
C02557=1074.347,217.696,419.152,174.221,26.936,154.752
C02558=1074.352,217.944,419.127,174.223,26.940,154.753
C02559=1074.358,218.193,419.101,174.225,26.944,154.753
C02560=1074.364,218.441,419.076,174.228,26.948,154.754
C02561=1074.370,218.690,419.050,174.230,26.952,154.754
C02562=1074.376,218.939,419.025,174.232,26.956,154.755
C02563=1074.382,219.187,419.000,174.234,26.959,154.755
C02564=1074.387,219.436,418.974,174.237,26.963,154.756
C02565=1074.393,219.685,418.948,174.239,26.967,154.757
C02566=1074.399,219.933,418.923,174.241,26.971,154.757
C02567=1074.405,220.182,418.897,174.243,26.975,154.758
C02568=1074.411,220.430,418.871,174.246,26.978,154.758
C02569=1074.416,220.679,418.846,174.247,26.982,154.759
C02570=1074.423,220.927,418.820,174.249,26.986,154.759
C02571=1074.429,221.176,418.795,174.251,26.990,154.760
C02572=1074.434,221.425,418.769,174.254,26.993,154.761
C02573=1074.444,221.844,418.726,174.257,27.000,154.762
C02574=1074.454,222.262,418.683,174.261,27.006,154.762
C02575=1074.464,222.681,418.639,174.265,27.013,154.764
C02576=1074.473,223.100,418.596,174.269,27.019,154.764
C02577=1074.479,223.349,418.570,174.271,27.023,154.765
C02578=1074.485,223.598,418.544,174.273,27.027,154.766
C02579=1074.490,223.845,418.518,174.275,27.030,154.766
C02580=1074.496,224.094,418.492,174.278,27.034,154.767
C02581=1074.502,224.343,418.467,174.280,27.038,154.767
C02582=1074.507,224.592,418.441,174.282,27.042,154.768
C02583=1074.513,224.840,418.414,174.284,27.046,154.768
C02584=1074.519,225.089,418.389,174.286,27.050,154.769
C02585=1074.525,225.338,418.363,174.289,27.053,154.770
C02586=1074.531,225.586,418.337,174.291,27.057,154.770
C02587=1074.537,225.835,418.311,174.293,27.061,154.771
C02588=1074.542,226.083,418.285,174.295,27.065,154.771
C02589=1074.548,226.331,418.259,174.298,27.069,154.772
C02590=1074.554,226.580,418.233,174.300,27.073,154.773
C02591=1074.559,226.829,418.208,174.302,27.076,154.773
C02592=1074.565,227.077,418.182,174.305,27.080,154.774
C02593=1074.571,227.326,418.156,174.307,27.084,154.774
C02594=1074.577,227.575,418.129,174.309,27.087,154.775
C02595=1074.583,227.823,418.104,174.311,27.091,154.775
C02596=1074.589,228.072,418.077,174.314,27.095,154.776
C02597=1074.594,228.321,418.051,174.316,27.099,154.776
C02598=1074.601,228.569,418.025,174.318,27.103,154.777
C02599=1074.606,228.818,417.999,174.320,27.106,154.778
C02600=1074.612,229.066,417.972,174.323,27.110,154.778
C02601=1074.617,229.315,417.946,174.325,27.114,154.779
C02602=1074.624,229.563,417.920,174.327,27.117,154.779
C02603=1074.629,229.812,417.894,174.329,27.121,154.780
C02604=1074.635,230.060,417.868,174.332,27.125,154.780
C02605=1074.641,230.309,417.842,174.334,27.129,154.781
C02606=1074.647,230.557,417.816,174.336,27.133,154.782
C02607=1074.653,230.806,417.790,174.338,27.137,154.782
C02608=1074.658,231.055,417.763,174.341,27.140,154.783
C02609=1074.664,231.303,417.737,174.343,27.144,154.783
C02610=1074.670,231.552,417.711,174.345,27.148,154.784
C02611=1074.675,231.800,417.684,174.347,27.152,154.785
C02612=1074.681,232.049,417.657,174.350,27.156,154.785
C02613=1074.687,232.298,417.631,174.352,27.159,154.786
C02614=1074.692,232.546,417.605,174.354,27.163,154.786
C02615=1074.700,232.795,417.578,174.357,27.167,154.787
C02616=1074.705,233.044,417.552,174.359,27.171,154.787
C02617=1074.711,233.292,417.526,174.361,27.174,154.788
C02618=1074.717,233.541,417.499,174.363,27.178,154.789
C02619=1074.722,233.789,417.472,174.366,27.182,154.789
C02620=1074.728,234.038,417.447,174.368,27.186,154.790
C02621=1074.734,234.286,417.420,174.371,27.190,154.790
C02622=1074.739,234.535,417.393,174.373,27.194,154.791
C02623=1074.745,234.783,417.367,174.376,27.198,154.791
C02624=1074.751,235.031,417.340,174.378,27.202,154.792
C02625=1074.760,235.442,417.296,174.382,27.208,154.793
C02626=1074.769,235.853,417.252,174.385,27.214,154.794
C02627=1074.779,236.263,417.208,174.389,27.220,154.795
C02628=1074.789,236.673,417.164,174.393,27.227,154.796
C02629=1074.795,236.922,417.138,174.395,27.230,154.796
C02630=1074.800,237.170,417.111,174.398,27.234,154.797
C02631=1074.806,237.419,417.084,174.400,27.238,154.798
C02632=1074.812,237.667,417.058,174.402,27.241,154.798
C02633=1074.818,237.916,417.031,174.404,27.245,154.799
C02634=1074.824,238.164,417.004,174.407,27.249,154.799
C02635=1074.830,238.413,416.977,174.409,27.253,154.800
C02636=1074.835,238.661,416.950,174.411,27.256,154.800
C02637=1074.841,238.910,416.923,174.414,27.261,154.801
C02638=1074.847,239.159,416.896,174.417,27.264,154.802
C02639=1074.853,239.407,416.870,174.419,27.268,154.802
C02640=1074.859,239.655,416.843,174.421,27.272,154.803
C02641=1074.864,239.904,416.816,174.424,27.276,154.803
C02642=1074.870,240.152,416.790,174.426,27.280,154.804
C02643=1074.877,240.401,416.763,174.428,27.283,154.804
C02644=1074.882,240.650,416.736,174.430,27.287,154.805
C02645=1074.887,240.898,416.709,174.433,27.291,154.806
C02646=1074.893,241.147,416.682,174.435,27.294,154.806
C02647=1074.899,241.395,416.656,174.437,27.298,154.807
C02648=1074.906,241.643,416.628,174.440,27.302,154.807
C02649=1074.911,241.892,416.601,174.442,27.306,154.808
C02650=1074.916,242.140,416.574,174.445,27.310,154.808
C02651=1074.923,242.390,416.547,174.448,27.313,154.809
C02652=1074.928,242.638,416.520,174.450,27.317,154.810
C02653=1074.935,242.886,416.493,174.452,27.321,154.810
C02654=1074.940,243.134,416.466,174.454,27.325,154.811
C02655=1074.946,243.383,416.439,174.457,27.328,154.811
C02656=1074.952,243.632,416.412,174.459,27.332,154.812
C02657=1074.957,243.880,416.384,174.461,27.336,154.812
C02658=1074.963,244.128,416.357,174.463,27.340,154.813
C02659=1074.969,244.377,416.330,174.467,27.344,154.814
C02660=1074.975,244.625,416.302,174.469,27.348,154.814
C02661=1074.980,244.874,416.276,174.471,27.351,154.815
C02662=1074.985,245.122,416.249,174.474,27.355,154.815
C02663=1074.992,245.371,416.221,174.476,27.359,154.816
C02664=1074.998,245.619,416.194,174.478,27.363,154.817
C02665=1075.003,245.868,416.167,174.480,27.367,154.817
C02666=1075.010,246.116,416.139,174.483,27.371,154.818
C02667=1075.015,246.365,416.112,174.486,27.374,154.818
C02668=1075.021,246.613,416.085,174.488,27.378,154.819
C02669=1075.027,246.862,416.058,174.491,27.382,154.819
C02670=1075.032,247.110,416.030,174.493,27.386,154.820
C02671=1075.037,247.358,416.002,174.495,27.390,154.821
C02672=1075.043,247.607,415.976,174.497,27.394,154.821
C02673=1075.049,247.856,415.947,174.500,27.397,154.822
C02674=1075.055,248.104,415.921,174.502,27.401,154.822
C02675=1075.060,248.352,415.893,174.505,27.405,154.823
C02676=1075.066,248.601,415.864,174.507,27.409,154.823
C02677=1075.075,249.004,415.820,174.511,27.415,154.824
C02678=1075.085,249.408,415.776,174.515,27.421,154.825
C02679=1075.094,249.812,415.731,174.519,27.428,154.826
C02680=1075.103,250.215,415.686,174.523,27.434,154.827
C02681=1075.109,250.465,415.659,174.525,27.438,154.828
C02682=1075.115,250.713,415.631,174.527,27.441,154.828
C02683=1075.120,250.961,415.603,174.531,27.446,154.829
C02684=1075.127,251.210,415.576,174.533,27.449,154.830
C02685=1075.132,251.458,415.548,174.535,27.453,154.830
C02686=1075.137,251.706,415.520,174.538,27.457,154.831
C02687=1075.144,251.955,415.493,174.540,27.461,154.831
C02688=1075.149,252.203,415.465,174.542,27.464,154.832
C02689=1075.155,252.452,415.436,174.545,27.469,154.833
C02690=1075.161,252.699,415.409,174.548,27.472,154.833
C02691=1075.167,252.949,415.382,174.550,27.476,154.834
C02692=1075.172,253.197,415.354,174.552,27.480,154.834
C02693=1075.178,253.445,415.326,174.555,27.484,154.835
C02694=1075.184,253.693,415.298,174.557,27.487,154.835
C02695=1075.189,253.941,415.270,174.560,27.492,154.836
C02696=1075.196,254.190,415.242,174.562,27.495,154.837
C02697=1075.201,254.438,415.215,174.565,27.499,154.837
C02698=1075.207,254.687,415.187,174.567,27.503,154.838
C02699=1075.212,254.935,415.159,174.569,27.507,154.838
C02700=1075.219,255.184,415.131,174.573,27.511,154.839
C02701=1075.224,255.432,415.103,174.575,27.515,154.840
C02702=1075.230,255.681,415.075,174.577,27.518,154.840
C02703=1075.236,255.929,415.047,174.580,27.522,154.841
C02704=1075.242,256.177,415.019,174.582,27.526,154.841
C02705=1075.248,256.425,414.991,174.585,27.530,154.842
C02706=1075.254,256.674,414.963,174.587,27.533,154.842
C02707=1075.260,256.922,414.935,174.590,27.537,154.843
C02708=1075.266,257.170,414.907,174.592,27.541,154.844
C02709=1075.272,257.419,414.879,174.594,27.544,154.844
C02710=1075.277,257.667,414.851,174.598,27.549,154.845
C02711=1075.283,257.916,414.822,174.600,27.552,154.845
C02712=1075.289,258.164,414.795,174.602,27.556,154.846
C02713=1075.295,258.412,414.767,174.605,27.560,154.846
C02714=1075.301,258.661,414.738,174.608,27.564,154.847
C02715=1075.306,258.909,414.710,174.610,27.568,154.848
C02716=1075.313,259.158,414.683,174.612,27.572,154.848
C02717=1075.318,259.406,414.655,174.615,27.575,154.849
C02718=1075.324,259.654,414.626,174.617,27.579,154.849
C02719=1075.330,259.903,414.598,174.620,27.583,154.850
C02720=1075.336,260.151,414.569,174.623,27.586,154.850
C02721=1075.342,260.399,414.542,174.625,27.590,154.851
C02722=1075.348,260.648,414.513,174.627,27.594,154.852
C02723=1075.354,260.896,414.485,174.631,27.598,154.852
C02724=1075.360,261.145,414.457,174.633,27.602,154.853
C02725=1075.366,261.393,414.428,174.635,27.606,154.853
C02726=1075.372,261.640,414.401,174.638,27.609,154.854
C02727=1075.378,261.889,414.372,174.641,27.613,154.854
C02728=1075.384,262.138,414.344,174.643,27.617,154.855
C02729=1075.393,262.539,414.298,174.647,27.623,154.856
C02730=1075.403,262.940,414.252,174.651,27.629,154.857
C02731=1075.413,263.341,414.207,174.656,27.635,154.858
C02732=1075.422,263.742,414.161,174.660,27.641,154.859
C02733=1075.428,263.990,414.132,174.662,27.645,154.859
C02734=1075.434,264.239,414.104,174.664,27.649,154.860
C02735=1075.440,264.487,414.075,174.668,27.653,154.860
C02736=1075.445,264.736,414.046,174.670,27.657,154.861
C02737=1075.452,264.984,414.017,174.672,27.661,154.862
C02738=1075.457,265.233,413.989,174.675,27.664,154.862
C02739=1075.463,265.481,413.961,174.678,27.669,154.863
C02740=1075.469,265.729,413.932,174.680,27.672,154.863
C02741=1075.475,265.978,413.903,174.683,27.676,154.864
C02742=1075.481,266.225,413.875,174.685,27.680,154.865
C02743=1075.486,266.474,413.846,174.688,27.684,154.865
C02744=1075.492,266.722,413.817,174.690,27.688,154.866
C02745=1075.498,266.970,413.788,174.693,27.691,154.866
C02746=1075.504,267.218,413.760,174.696,27.696,154.867
C02747=1075.510,267.466,413.731,174.698,27.699,154.868
C02748=1075.516,267.715,413.702,174.701,27.703,154.868
C02749=1075.521,267.964,413.673,174.703,27.707,154.869
C02750=1075.527,268.211,413.644,174.706,27.711,154.869
C02751=1075.533,268.460,413.616,174.709,27.715,154.870
C02752=1075.539,268.708,413.587,174.711,27.718,154.871
C02753=1075.545,268.957,413.558,174.714,27.723,154.871
C02754=1075.551,269.205,413.529,174.717,27.726,154.872
C02755=1075.556,269.453,413.500,174.719,27.730,154.872
C02756=1075.563,269.701,413.471,174.722,27.734,154.873
C02757=1075.569,269.949,413.443,174.724,27.738,154.874
C02758=1075.574,270.198,413.413,174.727,27.742,154.874
C02759=1075.580,270.446,413.384,174.729,27.745,154.875
C02760=1075.586,270.693,413.355,174.732,27.750,154.875
C02761=1075.591,270.943,413.326,174.735,27.754,154.876
C02762=1075.597,271.191,413.297,174.737,27.757,154.876
C02763=1075.604,271.439,413.268,174.740,27.761,154.877
C02764=1075.609,271.687,413.239,174.743,27.765,154.878
C02765=1075.615,271.935,413.210,174.745,27.769,154.878
C02766=1075.621,272.183,413.182,174.748,27.773,154.879
C02767=1075.626,272.432,413.152,174.751,27.777,154.879
C02768=1075.632,272.680,413.123,174.753,27.781,154.880
C02769=1075.639,272.928,413.094,174.756,27.785,154.881
C02770=1075.644,273.177,413.064,174.759,27.788,154.881
C02771=1075.650,273.425,413.035,174.761,27.792,154.882
C02772=1075.656,273.673,413.006,174.764,27.796,154.882
C02773=1075.662,273.921,412.977,174.766,27.800,154.883
C02774=1075.667,274.169,412.947,174.769,27.804,154.884
C02775=1075.673,274.417,412.918,174.772,27.808,154.884
C02776=1075.680,274.665,412.889,174.774,27.812,154.885
C02777=1075.685,274.914,412.860,174.777,27.816,154.886
C02778=1075.691,275.162,412.831,174.780,27.820,154.886
C02779=1075.697,275.410,412.801,174.782,27.824,154.887
C02780=1075.703,275.658,412.772,174.785,27.828,154.887
C02781=1075.712,276.063,412.724,174.790,27.834,154.888
C02782=1075.722,276.467,412.676,174.793,27.840,154.889
C02783=1075.731,276.872,412.628,174.798,27.847,154.890
C02784=1075.741,277.276,412.580,174.802,27.853,154.891
C02785=1075.746,277.524,412.550,174.804,27.857,154.892
C02786=1075.753,277.772,412.521,174.808,27.861,154.892
C02787=1075.758,278.021,412.492,174.810,27.865,154.893
C02788=1075.765,278.268,412.462,174.813,27.869,154.894
C02789=1075.770,278.517,412.432,174.816,27.873,154.894
C02790=1075.776,278.765,412.403,174.818,27.877,154.895
C02791=1075.782,279.013,412.374,174.821,27.881,154.896
C02792=1075.788,279.261,412.343,174.824,27.885,154.896
C02793=1075.794,279.509,412.314,174.826,27.888,154.897
C02794=1075.799,279.758,412.285,174.829,27.893,154.897
C02795=1075.805,280.006,412.255,174.832,27.897,154.898
C02796=1075.812,280.254,412.225,174.835,27.901,154.899
C02797=1075.817,280.502,412.196,174.837,27.904,154.899
C02798=1075.823,280.751,412.166,174.840,27.908,154.900
C02799=1075.829,280.998,412.136,174.843,27.912,154.900
C02800=1075.835,281.246,412.107,174.845,27.916,154.901
C02801=1075.840,281.494,412.076,174.848,27.920,154.902
C02802=1075.846,281.743,412.047,174.851,27.924,154.902
C02803=1075.851,281.991,412.017,174.853,27.928,154.903
C02804=1075.858,282.239,411.987,174.856,27.932,154.904
C02805=1075.864,282.487,411.958,174.859,27.936,154.904
C02806=1075.869,282.735,411.927,174.861,27.940,154.905
C02807=1075.875,282.983,411.898,174.864,27.944,154.905
C02808=1075.881,283.231,411.867,174.867,27.948,154.906
C02809=1075.887,283.479,411.838,174.870,27.952,154.907
C02810=1075.893,283.727,411.808,174.872,27.956,154.907
C02811=1075.899,283.976,411.778,174.875,27.960,154.908
C02812=1075.905,284.224,411.748,174.878,27.964,154.908
C02813=1075.910,284.472,411.717,174.880,27.968,154.909
C02814=1075.916,284.720,411.688,174.884,27.972,154.910
C02815=1075.922,284.968,411.657,174.886,27.976,154.910
C02816=1075.928,285.216,411.628,174.889,27.980,154.911
C02817=1075.934,285.464,411.598,174.891,27.984,154.912
C02818=1075.940,285.712,411.567,174.894,27.988,154.912
C02819=1075.945,285.960,411.538,174.897,27.992,154.913
C02820=1075.952,286.209,411.507,174.899,27.996,154.914
C02821=1075.957,286.457,411.477,174.903,28.000,154.914
C02822=1075.963,286.705,411.447,174.905,28.004,154.915
C02823=1075.969,286.953,411.417,174.908,28.009,154.915
C02824=1075.975,287.201,411.386,174.911,28.012,154.916
C02825=1075.981,287.448,411.357,174.913,28.016,154.917
C02826=1075.987,287.698,411.327,174.916,28.020,154.917
C02827=1075.993,287.945,411.296,174.919,28.024,154.918
C02828=1075.999,288.193,411.266,174.922,28.028,154.919
C02829=1076.005,288.441,411.236,174.924,28.032,154.919
C02830=1076.011,288.690,411.205,174.928,28.036,154.920
C02831=1076.017,288.938,411.175,174.930,28.040,154.920
C02832=1076.022,289.186,411.145,174.933,28.044,154.921
C02833=1076.032,289.599,411.094,174.937,28.051,154.922
C02834=1076.042,290.015,411.043,174.942,28.058,154.923
C02835=1076.052,290.429,410.993,174.947,28.065,154.924
C02836=1076.062,290.843,410.941,174.952,28.071,154.925
C02837=1076.068,291.091,410.911,174.954,28.075,154.926
C02838=1076.074,291.339,410.881,174.957,28.080,154.927
C02839=1076.080,291.586,410.850,174.960,28.084,154.927
C02840=1076.085,291.835,410.819,174.963,28.088,154.928
C02841=1076.091,292.083,410.789,174.965,28.092,154.929
C02842=1076.097,292.331,410.758,174.969,28.096,154.929
C02843=1076.103,292.579,410.728,174.971,28.100,154.930
C02844=1076.109,292.827,410.697,174.974,28.104,154.930
C02845=1076.115,293.075,410.667,174.977,28.108,154.931
C02846=1076.120,293.323,410.636,174.980,28.112,154.932
C02847=1076.127,293.572,410.605,174.982,28.116,154.932
C02848=1076.133,293.819,410.574,174.985,28.121,154.933
C02849=1076.138,294.067,410.544,174.988,28.125,154.934
C02850=1076.145,294.315,410.513,174.991,28.129,154.934
C02851=1076.150,294.563,410.482,174.993,28.133,154.935
C02852=1076.156,294.811,410.452,174.997,28.137,154.936
C02853=1076.162,295.059,410.420,174.999,28.141,154.936
C02854=1076.168,295.307,410.390,175.002,28.145,154.937
C02855=1076.173,295.555,410.359,175.005,28.149,154.938
C02856=1076.180,295.804,410.328,175.008,28.153,154.938
C02857=1076.186,296.051,410.297,175.010,28.157,154.939
C02858=1076.192,296.299,410.267,175.014,28.161,154.940
C02859=1076.197,296.548,410.236,175.016,28.165,154.940
C02860=1076.204,296.795,410.204,175.019,28.170,154.941
C02861=1076.209,297.043,410.174,175.022,28.174,154.941
C02862=1076.215,297.291,410.143,175.025,28.178,154.942
C02863=1076.221,297.539,410.112,175.027,28.182,154.943
C02864=1076.227,297.787,410.080,175.031,28.186,154.943
C02865=1076.233,298.035,410.050,175.033,28.190,154.944
C02866=1076.238,298.283,410.018,175.036,28.195,154.945
C02867=1076.244,298.531,409.988,175.039,28.199,154.945
C02868=1076.250,298.779,409.956,175.042,28.203,154.946
C02869=1076.256,299.027,409.926,175.044,28.207,154.947
C02870=1076.262,299.275,409.894,175.047,28.211,154.948
C02871=1076.267,299.523,409.863,175.051,28.216,154.948
C02872=1076.273,299.770,409.832,175.053,28.220,154.949
C02873=1076.279,300.019,409.800,175.056,28.224,154.950
C02874=1076.285,300.266,409.769,175.059,28.228,154.950
C02875=1076.291,300.514,409.737,175.062,28.232,154.951
C02876=1076.296,300.762,409.707,175.064,28.237,154.952
C02877=1076.302,301.010,409.675,175.068,28.241,154.952
C02878=1076.308,301.259,409.644,175.070,28.245,154.953
C02879=1076.314,301.506,409.613,175.073,28.249,154.954
C02880=1076.320,301.754,409.581,175.076,28.254,154.954
C02881=1076.325,302.002,409.550,175.079,28.258,154.955
C02882=1076.331,302.250,409.518,175.082,28.262,154.956
C02883=1076.337,302.498,409.487,175.084,28.267,154.956
C02884=1076.343,302.746,409.456,175.088,28.271,154.957
C02885=1076.347,302.960,409.428,175.090,28.274,154.958
C02886=1076.353,303.175,409.401,175.093,28.278,154.958
C02887=1076.358,303.388,409.374,175.095,28.281,154.959
C02888=1076.363,303.603,409.347,175.097,28.285,154.960
C02889=1076.368,303.818,409.319,175.100,28.289,154.960
C02890=1076.373,304.032,409.293,175.102,28.293,154.961
C02891=1076.379,304.246,409.265,175.106,28.296,154.961
C02892=1076.383,304.462,409.238,175.108,28.300,154.962
C02893=1076.389,304.709,409.207,175.110,28.304,154.963
C02894=1076.395,304.957,409.175,175.114,28.308,154.963
C02895=1076.401,305.204,409.143,175.116,28.313,154.964
C02896=1076.407,305.452,409.112,175.119,28.317,154.965
C02897=1076.413,305.700,409.080,175.123,28.321,154.965
C02898=1076.419,305.948,409.048,175.125,28.326,154.966
C02899=1076.426,306.196,409.016,175.128,28.330,154.967
C02900=1076.431,306.444,408.986,175.132,28.334,154.967
C02901=1076.437,306.692,408.953,175.134,28.339,154.968
C02902=1076.442,306.940,408.922,175.137,28.343,154.969
C02903=1076.449,307.188,408.890,175.140,28.347,154.969
C02904=1076.455,307.436,408.858,175.143,28.351,154.970
C02905=1076.460,307.683,408.827,175.146,28.356,154.971
C02906=1076.467,307.931,408.795,175.148,28.360,154.972
C02907=1076.473,308.179,408.763,175.152,28.364,154.972
C02908=1076.478,308.426,408.731,175.155,28.368,154.973
C02909=1076.484,308.675,408.699,175.157,28.373,154.974
C02910=1076.491,308.923,408.667,175.161,28.377,154.974
C02911=1076.497,309.170,408.636,175.163,28.381,154.975
C02912=1076.503,309.418,408.604,175.166,28.386,154.976
C02913=1076.509,309.667,408.572,175.170,28.390,154.976
C02914=1076.514,309.914,408.540,175.172,28.394,154.977
C02915=1076.521,310.162,408.509,175.175,28.398,154.978
C02916=1076.527,310.410,408.476,175.179,28.403,154.978
C02917=1076.533,310.658,408.444,175.181,28.407,154.979
C02918=1076.538,310.905,408.412,175.184,28.411,154.980
C02919=1076.544,311.153,408.380,175.187,28.416,154.981
C02920=1076.551,311.401,408.348,175.190,28.420,154.981
C02921=1076.557,311.649,408.316,175.193,28.425,154.982
C02922=1076.563,311.896,408.284,175.196,28.429,154.983
C02923=1076.569,312.145,408.252,175.199,28.433,154.983
C02924=1076.575,312.392,408.220,175.202,28.437,154.984
C02925=1076.582,312.640,408.188,175.205,28.441,154.985
C02926=1076.588,312.888,408.156,175.208,28.446,154.986
C02927=1076.594,313.136,408.123,175.211,28.450,154.986
C02928=1076.599,313.384,408.092,175.214,28.455,154.987
C02929=1076.605,313.632,408.060,175.217,28.459,154.988
C02930=1076.612,313.879,408.027,175.220,28.463,154.988
C02931=1076.618,314.128,407.995,175.223,28.468,154.989
C02932=1076.625,314.375,407.963,175.226,28.472,154.990
C02933=1076.631,314.623,407.931,175.229,28.476,154.990
C02934=1076.636,314.871,407.897,175.232,28.481,154.991
C02935=1076.642,315.118,407.866,175.235,28.485,154.992
C02936=1076.648,315.366,407.833,175.238,28.489,154.993
C02937=1076.654,315.614,407.801,175.241,28.494,154.993
C02938=1076.659,315.862,407.768,175.244,28.499,154.994
C02939=1076.665,316.110,407.736,175.247,28.503,154.995
C02940=1076.671,316.357,407.703,175.250,28.508,154.996
C02941=1076.675,316.574,407.675,175.252,28.512,154.996
C02942=1076.681,316.790,407.646,175.255,28.516,154.997
C02943=1076.687,317.006,407.618,175.258,28.520,154.998
C02944=1076.691,317.222,407.589,175.261,28.524,154.998
C02945=1076.696,317.438,407.562,175.263,28.528,154.999
C02946=1076.702,317.654,407.533,175.265,28.532,155.000
C02947=1076.706,317.870,407.504,175.268,28.535,155.000
C02948=1076.712,318.086,407.475,175.271,28.540,155.001
C02949=1076.718,318.334,407.443,175.274,28.543,155.002
C02950=1076.723,318.582,407.410,175.277,28.548,155.002
C02951=1076.730,318.829,407.377,175.280,28.553,155.003
C02952=1076.736,319.077,407.345,175.283,28.558,155.004
C02953=1076.741,319.325,407.312,175.286,28.562,155.005
C02954=1076.747,319.572,407.280,175.289,28.567,155.006
C02955=1076.752,319.820,407.246,175.292,28.571,155.006
C02956=1076.759,320.068,407.214,175.295,28.576,155.007
C02957=1076.765,320.315,407.181,175.298,28.580,155.008
C02958=1076.770,320.564,407.148,175.301,28.585,155.009
C02959=1076.777,320.811,407.115,175.305,28.589,155.009
C02960=1076.783,321.059,407.083,175.307,28.594,155.010
C02961=1076.788,321.307,407.049,175.310,28.598,155.011
C02962=1076.795,321.555,407.017,175.313,28.603,155.012
C02963=1076.800,321.802,406.983,175.317,28.608,155.012
C02964=1076.807,322.050,406.951,175.319,28.612,155.013
C02965=1076.813,322.298,406.918,175.322,28.617,155.014
C02966=1076.818,322.546,406.884,175.326,28.621,155.015
C02967=1076.825,322.793,406.852,175.329,28.626,155.015
C02968=1076.830,323.041,406.818,175.331,28.630,155.016
C02969=1076.837,323.289,406.786,175.335,28.635,155.017
C02970=1076.842,323.537,406.752,175.338,28.640,155.018
C02971=1076.848,323.784,406.720,175.341,28.644,155.019
C02972=1076.855,324.032,406.687,175.344,28.649,155.019
C02973=1076.860,324.280,406.653,175.347,28.653,155.020
C02974=1076.867,324.528,406.620,175.350,28.658,155.021
C02975=1076.873,324.776,406.587,175.353,28.663,155.022
C02976=1076.879,325.023,406.554,175.357,28.667,155.022
C02977=1076.885,325.271,406.520,175.359,28.672,155.023
C02978=1076.891,325.518,406.487,175.362,28.676,155.024
C02979=1076.897,325.766,406.454,175.366,28.681,155.025
C02980=1076.903,326.014,406.421,175.369,28.686,155.026
C02981=1076.909,326.262,406.388,175.372,28.691,155.026
C02982=1076.916,326.509,406.354,175.375,28.695,155.027
C02983=1076.921,326.757,406.321,175.378,28.700,155.028
C02984=1076.928,327.005,406.288,175.381,28.705,155.029
C02985=1076.933,327.253,406.255,175.384,28.709,155.030
C02986=1076.940,327.500,406.221,175.388,28.714,155.030
C02987=1076.946,327.748,406.188,175.390,28.718,155.031
C02988=1076.952,327.996,406.155,175.393,28.723,155.032
C02989=1076.958,328.243,406.121,175.397,28.728,155.033
C02990=1076.964,328.491,406.088,175.400,28.733,155.034
C02991=1076.970,328.739,406.055,175.403,28.737,155.034
C02992=1076.977,328.986,406.021,175.407,28.742,155.035
C02993=1076.983,329.234,405.988,175.409,28.746,155.036
C02994=1076.989,329.482,405.954,175.412,28.751,155.037
C02995=1076.995,329.729,405.921,175.416,28.756,155.038
C02996=1077.001,329.978,405.887,175.419,28.761,155.038
C02997=1077.007,330.190,405.858,175.421,28.765,155.039
C02998=1077.011,330.403,405.829,175.425,28.769,155.040
C02999=1077.018,330.616,405.800,175.427,28.773,155.040
C03000=1077.023,330.829,405.772,175.429,28.777,155.041
C03001=1077.028,331.041,405.743,175.433,28.781,155.042
C03002=1077.033,331.254,405.714,175.435,28.785,155.042
C03003=1077.039,331.467,405.684,175.438,28.789,155.043
C03004=1077.044,331.680,405.656,175.441,28.794,155.044
C03005=1077.050,331.927,405.622,175.443,28.798,155.045
C03006=1077.056,332.175,405.588,175.447,28.803,155.046
C03007=1077.061,332.423,405.555,175.450,28.808,155.046
C03008=1077.068,332.671,405.521,175.453,28.813,155.047
C03009=1077.074,332.918,405.487,175.457,28.817,155.048
C03010=1077.079,333.166,405.453,175.460,28.823,155.049
C03011=1077.086,333.414,405.419,175.463,28.827,155.050
C03012=1077.092,333.661,405.385,175.466,28.832,155.051
C03013=1077.098,333.908,405.351,175.469,28.837,155.051
C03014=1077.104,334.157,405.318,175.472,28.842,155.052
C03015=1077.110,334.404,405.284,175.475,28.847,155.053
C03016=1077.116,334.651,405.249,175.479,28.852,155.054
C03017=1077.122,334.899,405.215,175.482,28.857,155.055
C03018=1077.128,335.147,405.181,175.485,28.861,155.056
C03019=1077.134,335.394,405.147,175.488,28.867,155.057
C03020=1077.140,335.642,405.113,175.492,28.871,155.057
C03021=1077.146,335.890,405.079,175.495,28.876,155.058
C03022=1077.153,336.138,405.045,175.498,28.881,155.059
C03023=1077.158,336.385,405.011,175.502,28.886,155.060
C03024=1077.164,336.632,404.977,175.504,28.891,155.061
C03025=1077.171,336.880,404.942,175.507,28.896,155.062
C03026=1077.177,337.128,404.908,175.511,28.901,155.062
C03027=1077.183,337.376,404.874,175.514,28.906,155.063
C03028=1077.189,337.623,404.840,175.517,28.911,155.064
C03029=1077.195,337.871,404.805,175.520,28.916,155.065
C03030=1077.201,338.118,404.771,175.524,28.921,155.066
C03031=1077.207,338.365,404.737,175.527,28.926,155.067
C03032=1077.214,338.613,404.703,175.530,28.931,155.068
C03033=1077.219,338.861,404.669,175.534,28.936,155.069
C03034=1077.226,339.108,404.634,175.537,28.941,155.070
C03035=1077.232,339.355,404.600,175.540,28.946,155.070
C03036=1077.238,339.604,404.565,175.543,28.951,155.071
C03037=1077.244,339.851,404.530,175.547,28.956,155.072
C03038=1077.250,340.099,404.496,175.550,28.961,155.073
C03039=1077.256,340.346,404.462,175.553,28.966,155.074
C03040=1077.263,340.593,404.427,175.557,28.971,155.075
C03041=1077.268,340.841,404.392,175.560,28.977,155.076
C03042=1077.274,341.089,404.358,175.563,28.982,155.077
C03043=1077.280,341.336,404.323,175.566,28.987,155.077
C03044=1077.287,341.584,404.289,175.570,28.992,155.078
C03045=1077.293,341.831,404.255,175.572,28.997,155.079
C03046=1077.299,342.079,404.220,175.575,29.002,155.080
C03047=1077.305,342.326,404.185,175.579,29.007,155.081
C03048=1077.311,342.574,404.150,175.582,29.012,155.082
C03049=1077.318,342.821,404.115,175.585,29.017,155.083
C03050=1077.323,343.069,404.081,175.588,29.022,155.084
C03051=1077.330,343.317,404.046,175.592,29.027,155.085
C03052=1077.336,343.564,404.011,175.596,29.033,155.086
C03053=1077.341,343.774,403.982,175.598,29.037,155.086
C03054=1077.346,343.984,403.952,175.601,29.041,155.087
C03055=1077.352,344.194,403.922,175.604,29.046,155.088
C03056=1077.357,344.405,403.893,175.607,29.050,155.089
C03057=1077.361,344.615,403.863,175.610,29.055,155.090
C03058=1077.367,344.825,403.834,175.612,29.059,155.090
C03059=1077.372,345.035,403.804,175.615,29.064,155.091
C03060=1077.378,345.245,403.774,175.618,29.068,155.092
C03061=1077.384,345.492,403.740,175.621,29.073,155.093
C03062=1077.389,345.740,403.705,175.625,29.079,155.094
C03063=1077.396,345.988,403.670,175.628,29.084,155.095
C03064=1077.402,346.235,403.634,175.631,29.089,155.096
C03065=1077.408,346.483,403.600,175.634,29.095,155.097
C03066=1077.414,346.730,403.564,175.638,29.100,155.098
C03067=1077.420,346.977,403.529,175.641,29.105,155.099
C03068=1077.426,347.225,403.494,175.644,29.111,155.100
C03069=1077.433,347.473,403.459,175.648,29.116,155.100
C03070=1077.438,347.720,403.424,175.651,29.121,155.101
C03071=1077.445,347.967,403.389,175.654,29.126,155.102
C03072=1077.451,348.215,403.353,175.657,29.132,155.103
C03073=1077.457,348.461,403.318,175.661,29.137,155.104
C03074=1077.463,348.710,403.283,175.665,29.143,155.105
C03075=1077.470,348.957,403.248,175.668,29.148,155.106
C03076=1077.476,349.205,403.212,175.671,29.154,155.107
C03077=1077.481,349.452,403.177,175.675,29.159,155.108
C03078=1077.488,349.699,403.142,175.678,29.164,155.109
C03079=1077.494,349.947,403.106,175.681,29.169,155.110
C03080=1077.501,350.194,403.071,175.685,29.175,155.111
C03081=1077.506,350.441,403.036,175.688,29.181,155.112
C03082=1077.512,350.689,403.000,175.691,29.186,155.113
C03083=1077.519,350.936,402.965,175.694,29.191,155.114
C03084=1077.525,351.184,402.929,175.698,29.196,155.115
C03085=1077.532,351.431,402.894,175.702,29.202,155.116
C03086=1077.537,351.678,402.858,175.705,29.208,155.117
C03087=1077.543,351.926,402.823,175.709,29.213,155.118
C03088=1077.550,352.173,402.788,175.712,29.218,155.119
C03089=1077.556,352.421,402.752,175.715,29.224,155.120
C03090=1077.562,352.668,402.716,175.718,29.230,155.121
C03091=1077.569,352.915,402.680,175.722,29.235,155.122
C03092=1077.575,353.162,402.645,175.725,29.240,155.123
C03093=1077.581,353.410,402.609,175.729,29.246,155.124
C03094=1077.587,353.658,402.573,175.732,29.252,155.125
C03095=1077.593,353.905,402.538,175.736,29.257,155.126
C03096=1077.600,354.152,402.502,175.739,29.263,155.127
C03097=1077.606,354.400,402.466,175.742,29.268,155.128
C03098=1077.612,354.647,402.430,175.746,29.274,155.129
C03099=1077.617,354.894,402.394,175.749,29.279,155.130
C03100=1077.624,355.141,402.359,175.753,29.285,155.131
C03101=1077.630,355.389,402.323,175.756,29.291,155.132
C03102=1077.636,355.636,402.286,175.760,29.296,155.133
C03103=1077.643,355.883,402.251,175.763,29.302,155.134
C03104=1077.649,356.130,402.215,175.766,29.308,155.135
C03105=1077.655,356.378,402.179,175.769,29.313,155.136
C03106=1077.661,356.625,402.143,175.774,29.319,155.137
C03107=1077.667,356.873,402.107,175.777,29.325,155.138
C03108=1077.673,357.121,402.071,175.780,29.331,155.140
C03109=1077.679,357.332,402.040,175.784,29.336,155.140
C03110=1077.684,357.543,402.010,175.786,29.340,155.141
C03111=1077.690,357.756,401.978,175.789,29.345,155.142
C03112=1077.695,357.967,401.947,175.792,29.350,155.143
C03113=1077.700,358.179,401.917,175.795,29.355,155.144
C03114=1077.705,358.390,401.885,175.798,29.360,155.145
C03115=1077.711,358.602,401.854,175.801,29.365,155.146
C03116=1077.717,358.814,401.823,175.804,29.370,155.147
C03117=1077.723,359.062,401.788,175.807,29.375,155.148
C03118=1077.729,359.309,401.751,175.811,29.381,155.149
C03119=1077.735,359.556,401.715,175.814,29.387,155.150
C03120=1077.741,359.803,401.679,175.818,29.393,155.151
C03121=1077.748,360.050,401.643,175.822,29.399,155.152
C03122=1077.754,360.297,401.606,175.825,29.404,155.153
C03123=1077.760,360.544,401.570,175.828,29.410,155.154
C03124=1077.766,360.792,401.534,175.831,29.416,155.155
C03125=1077.772,361.040,401.497,175.836,29.422,155.156
C03126=1077.778,361.287,401.461,175.839,29.428,155.158
C03127=1077.785,361.534,401.424,175.842,29.434,155.159
C03128=1077.792,361.781,401.387,175.845,29.439,155.160
C03129=1077.798,362.028,401.351,175.850,29.446,155.161
C03130=1077.804,362.276,401.314,175.853,29.451,155.162
C03131=1077.811,362.523,401.278,175.856,29.457,155.163
C03132=1077.817,362.770,401.242,175.859,29.463,155.164
C03133=1077.823,363.017,401.206,175.864,29.469,155.165
C03134=1077.829,363.265,401.169,175.867,29.475,155.166
C03135=1077.835,363.512,401.132,175.870,29.481,155.168
C03136=1077.842,363.759,401.096,175.874,29.488,155.169
C03137=1077.849,364.006,401.058,175.878,29.493,155.170
C03138=1077.855,364.253,401.022,175.881,29.499,155.171
C03139=1077.861,364.500,400.985,175.884,29.505,155.172
C03140=1077.867,364.747,400.948,175.889,29.512,155.173
C03141=1077.874,364.995,400.912,175.892,29.518,155.174
C03142=1077.880,365.242,400.875,175.895,29.524,155.175
C03143=1077.886,365.490,400.838,175.899,29.530,155.177
C03144=1077.892,365.736,400.801,175.903,29.536,155.178
C03145=1077.898,365.983,400.764,175.906,29.542,155.179
C03146=1077.904,366.230,400.728,175.909,29.548,155.180
C03147=1077.911,366.478,400.691,175.913,29.554,155.181
C03148=1077.917,366.725,400.653,175.917,29.560,155.182
C03149=1077.923,366.972,400.616,175.920,29.566,155.184
C03150=1077.929,367.219,400.579,175.924,29.573,155.185
C03151=1077.936,367.466,400.542,175.927,29.579,155.186
C03152=1077.942,367.714,400.505,175.931,29.585,155.187
C03153=1077.948,367.961,400.468,175.935,29.591,155.188
C03154=1077.955,368.207,400.431,175.938,29.597,155.189
C03155=1077.961,368.455,400.394,175.941,29.603,155.191
C03156=1077.968,368.702,400.357,175.946,29.610,155.192
C03157=1077.973,368.949,400.320,175.949,29.616,155.193
C03158=1077.980,369.196,400.283,175.952,29.622,155.194
C03159=1077.986,369.444,400.245,175.956,29.629,155.195
C03160=1077.993,369.690,400.208,175.960,29.635,155.197
C03161=1077.998,369.937,400.171,175.964,29.641,155.198
C03162=1078.006,370.185,400.133,175.967,29.648,155.199
C03163=1078.012,370.431,400.096,175.970,29.654,155.200
C03164=1078.018,370.678,400.059,175.975,29.661,155.202
C03165=1078.024,370.899,400.025,175.978,29.666,155.203
C03166=1078.030,371.119,399.992,175.980,29.671,155.204
C03167=1078.035,371.338,399.959,175.984,29.677,155.205
C03168=1078.041,371.559,399.926,175.987,29.683,155.206
C03169=1078.047,371.778,399.893,175.990,29.689,155.207
C03170=1078.052,371.998,399.859,175.994,29.694,155.208
C03171=1078.059,372.218,399.826,175.997,29.700,155.209
C03172=1078.064,372.438,399.792,176.000,29.706,155.210
C03173=1078.070,372.685,399.755,176.004,29.712,155.212
C03174=1078.076,372.933,399.717,176.008,29.719,155.213
C03175=1078.083,373.179,399.680,176.011,29.725,155.214
C03176=1078.090,373.427,399.642,176.015,29.732,155.215
C03177=1078.096,373.673,399.605,176.019,29.738,155.216
C03178=1078.103,373.921,399.567,176.022,29.744,155.218
C03179=1078.109,374.167,399.529,176.026,29.751,155.219
C03180=1078.114,374.414,399.491,176.029,29.758,155.220
C03181=1078.121,374.661,399.453,176.034,29.764,155.222
C03182=1078.128,374.908,399.416,176.037,29.771,155.223
C03183=1078.134,375.155,399.378,176.041,29.778,155.224
C03184=1078.140,375.402,399.340,176.044,29.784,155.225
C03185=1078.147,375.650,399.302,176.048,29.791,155.227
C03186=1078.152,375.896,399.264,176.052,29.798,155.228
C03187=1078.160,376.143,399.227,176.055,29.804,155.229
C03188=1078.166,376.390,399.189,176.059,29.811,155.231
C03189=1078.172,376.638,399.151,176.063,29.818,155.232
C03190=1078.178,376.884,399.112,176.067,29.824,155.233
C03191=1078.185,377.131,399.074,176.070,29.831,155.235
C03192=1078.191,377.378,399.036,176.074,29.838,155.236
C03193=1078.197,377.625,398.998,176.078,29.845,155.237
C03194=1078.204,377.871,398.960,176.082,29.852,155.239
C03195=1078.211,378.119,398.922,176.085,29.858,155.240
C03196=1078.217,378.366,398.884,176.089,29.865,155.241
C03197=1078.223,378.613,398.846,176.093,29.872,155.243
C03198=1078.230,378.860,398.808,176.097,29.879,155.244
C03199=1078.236,379.106,398.770,176.100,29.886,155.245
C03200=1078.243,379.353,398.731,176.104,29.892,155.247
C03201=1078.249,379.601,398.693,176.108,29.899,155.248
C03202=1078.255,379.847,398.655,176.112,29.906,155.249
C03203=1078.263,380.094,398.617,176.115,29.913,155.251
C03204=1078.269,380.341,398.579,176.119,29.920,155.252
C03205=1078.275,380.587,398.540,176.123,29.927,155.253
C03206=1078.282,380.835,398.502,176.127,29.934,155.255
C03207=1078.289,381.082,398.463,176.130,29.940,155.256
C03208=1078.295,381.329,398.425,176.135,29.948,155.257
C03209=1078.301,381.575,398.387,176.139,29.955,155.259
C03210=1078.308,381.822,398.348,176.142,29.962,155.260
C03211=1078.315,382.070,398.310,176.146,29.968,155.262
C03212=1078.321,382.316,398.271,176.150,29.975,155.263
C03213=1078.327,382.563,398.232,176.154,29.983,155.264
C03214=1078.333,382.810,398.194,176.157,29.990,155.266
C03215=1078.340,383.056,398.155,176.161,29.997,155.267
C03216=1078.346,383.303,398.116,176.165,30.004,155.269
C03217=1078.353,383.550,398.078,176.169,30.011,155.270
C03218=1078.359,383.797,398.038,176.173,30.019,155.272
C03219=1078.365,384.044,398.000,176.176,30.026,155.273
C03220=1078.372,384.291,397.962,176.181,30.033,155.274
C03221=1078.378,384.525,397.925,176.184,30.040,155.276
C03222=1078.384,384.759,397.887,176.188,30.047,155.277
C03223=1078.391,384.994,397.851,176.191,30.053,155.278
C03224=1078.397,385.228,397.814,176.195,30.060,155.280
C03225=1078.403,385.462,397.776,176.199,30.067,155.281
C03226=1078.409,385.696,397.740,176.202,30.074,155.283
C03227=1078.415,385.931,397.703,176.207,30.081,155.284
C03228=1078.421,386.165,397.666,176.210,30.088,155.285
C03229=1078.428,386.412,397.628,176.214,30.096,155.287
C03230=1078.435,386.659,397.587,176.217,30.103,155.288
C03231=1078.441,386.906,397.549,176.222,30.110,155.290
C03232=1078.448,387.152,397.510,176.226,30.117,155.291
C03233=1078.454,387.399,397.470,176.229,30.125,155.293
C03234=1078.460,387.646,397.432,176.233,30.133,155.294
C03235=1078.467,387.892,397.393,176.238,30.140,155.296
C03236=1078.473,388.140,397.354,176.241,30.147,155.297
C03237=1078.480,388.386,397.314,176.245,30.155,155.299
C03238=1078.487,388.633,397.275,176.249,30.163,155.300
C03239=1078.493,388.880,397.236,176.253,30.169,155.302
C03240=1078.500,389.127,397.197,176.257,30.177,155.303
C03241=1078.507,389.373,397.157,176.261,30.185,155.305
C03242=1078.513,389.620,397.118,176.264,30.192,155.306
C03243=1078.520,389.866,397.078,176.269,30.200,155.308
C03244=1078.527,390.113,397.040,176.273,30.207,155.310
C03245=1078.533,390.360,397.000,176.277,30.215,155.311
C03246=1078.540,390.606,396.961,176.280,30.223,155.313
C03247=1078.547,390.853,396.922,176.285,30.230,155.314
C03248=1078.554,391.100,396.882,176.289,30.238,155.316
C03249=1078.561,391.346,396.843,176.293,30.245,155.317
C03250=1078.567,391.593,396.803,176.296,30.253,155.319
C03251=1078.574,391.840,396.763,176.301,30.261,155.320
C03252=1078.581,392.087,396.723,176.305,30.269,155.322
C03253=1078.587,392.333,396.683,176.309,30.277,155.324
C03254=1078.594,392.580,396.644,176.313,30.284,155.325
C03255=1078.600,392.827,396.604,176.317,30.292,155.327
C03256=1078.607,393.073,396.565,176.321,30.300,155.328
C03257=1078.613,393.320,396.525,176.325,30.308,155.330
C03258=1078.620,393.567,396.485,176.329,30.316,155.332
C03259=1078.627,393.813,396.445,176.333,30.324,155.333
C03260=1078.634,394.061,396.406,176.337,30.332,155.335
C03261=1078.640,394.307,396.365,176.341,30.339,155.336
C03262=1078.647,394.553,396.326,176.346,30.347,155.338
C03263=1078.653,394.800,396.286,176.349,30.355,155.340
C03264=1078.660,395.046,396.246,176.353,30.363,155.341
C03265=1078.666,395.293,396.205,176.357,30.372,155.343
C03266=1078.674,395.540,396.166,176.362,30.380,155.345
C03267=1078.680,395.786,396.125,176.366,30.388,155.346
C03268=1078.687,396.033,396.085,176.369,30.396,155.348
C03269=1078.693,396.279,396.045,176.373,30.404,155.350
C03270=1078.700,396.527,396.005,176.378,30.412,155.351
C03271=1078.707,396.773,395.965,176.382,30.420,155.353
C03272=1078.714,397.019,395.925,176.386,30.428,155.355
C03273=1078.720,397.266,395.885,176.391,30.437,155.357
C03274=1078.727,397.513,395.844,176.394,30.445,155.358
C03275=1078.733,397.760,395.804,176.398,30.453,155.360
C03276=1078.740,398.006,395.764,176.402,30.461,155.362
C03277=1078.746,398.230,395.727,176.407,30.469,155.363
C03278=1078.752,398.455,395.690,176.410,30.476,155.365
C03279=1078.758,398.679,395.654,176.413,30.484,155.366
C03280=1078.765,398.903,395.617,176.418,30.491,155.368
C03281=1078.771,399.127,395.580,176.421,30.499,155.369
C03282=1078.777,399.352,395.544,176.425,30.507,155.371
C03283=1078.783,399.575,395.507,176.429,30.514,155.373
C03284=1078.789,399.800,395.470,176.433,30.522,155.374
C03285=1078.796,400.046,395.429,176.437,30.530,155.376
C03286=1078.803,400.293,395.388,176.441,30.539,155.378
C03287=1078.809,400.539,395.348,176.445,30.547,155.380
C03288=1078.816,400.786,395.307,176.449,30.556,155.381
C03289=1078.823,401.033,395.267,176.453,30.564,155.383
C03290=1078.830,401.279,395.226,176.458,30.573,155.385
C03291=1078.836,401.526,395.186,176.462,30.581,155.387
C03292=1078.844,401.772,395.144,176.466,30.590,155.389
C03293=1078.850,402.019,395.104,176.471,30.599,155.390
C03294=1078.857,402.265,395.063,176.475,30.607,155.392
C03295=1078.864,402.511,395.022,176.479,30.616,155.394
C03296=1078.871,402.759,394.982,176.483,30.625,155.396
C03297=1078.877,403.005,394.940,176.488,30.633,155.398
C03298=1078.884,403.252,394.900,176.492,30.642,155.399
C03299=1078.890,403.498,394.859,176.496,30.651,155.401
C03300=1078.898,403.744,394.817,176.501,30.659,155.403
C03301=1078.905,403.991,394.776,176.505,30.668,155.405
C03302=1078.911,404.238,394.736,176.509,30.677,155.407
C03303=1078.918,404.484,394.694,176.513,30.686,155.409
C03304=1078.925,404.730,394.653,176.518,30.695,155.411
C03305=1078.932,404.977,394.612,176.522,30.704,155.412
C03306=1078.939,405.224,394.570,176.526,30.713,155.414
C03307=1078.945,405.470,394.530,176.531,30.722,155.416
C03308=1078.952,405.716,394.488,176.535,30.731,155.418
C03309=1078.959,405.963,394.446,176.539,30.740,155.420
C03310=1078.966,406.209,394.406,176.544,30.749,155.422
C03311=1078.973,406.456,394.364,176.549,30.758,155.424
C03312=1078.980,406.703,394.323,176.553,30.767,155.426
C03313=1078.986,406.949,394.282,176.557,30.776,155.428
C03314=1078.994,407.195,394.240,176.562,30.786,155.430
C03315=1079.000,407.442,394.199,176.566,30.795,155.432
C03316=1079.007,407.689,394.157,176.570,30.804,155.434
C03317=1079.014,407.934,394.115,176.575,30.813,155.436
C03318=1079.021,408.181,394.074,176.579,30.822,155.438
C03319=1079.027,408.428,394.032,176.583,30.832,155.440
C03320=1079.034,408.675,393.990,176.589,30.841,155.442
C03321=1079.042,408.956,393.943,176.593,30.851,155.444
C03322=1079.050,409.236,393.896,176.598,30.862,155.446
C03323=1079.058,409.518,393.847,176.603,30.873,155.449
C03324=1079.065,409.799,393.800,176.608,30.884,155.451
C03325=1079.073,410.045,393.758,176.613,30.893,155.453
C03326=1079.080,410.292,393.716,176.618,30.903,155.455
C03327=1079.086,410.538,393.674,176.622,30.912,155.457
C03328=1079.093,410.784,393.633,176.627,30.922,155.459
C03329=1079.100,411.031,393.590,176.631,30.932,155.461
C03330=1079.107,411.277,393.549,176.636,30.941,155.463
C03331=1079.114,411.523,393.507,176.641,30.951,155.465
C03332=1079.121,411.770,393.464,176.645,30.960,155.467
C03333=1079.128,412.013,393.423,176.649,30.970,155.469
C03334=1079.135,412.256,393.382,176.654,30.979,155.471
C03335=1079.142,412.498,393.341,176.659,30.989,155.474
C03336=1079.149,412.742,393.299,176.663,30.998,155.476
C03337=1079.156,412.984,393.257,176.668,31.008,155.478
C03338=1079.162,413.227,393.216,176.672,31.018,155.480
C03339=1079.170,413.469,393.174,176.677,31.027,155.482
C03340=1079.177,413.711,393.133,176.682,31.037,155.484
C03341=1079.184,413.958,393.090,176.686,31.047,155.486
C03342=1079.190,414.205,393.048,176.690,31.057,155.488
C03343=1079.198,414.452,393.005,176.696,31.067,155.490
C03344=1079.205,414.698,392.963,176.700,31.077,155.493
C03345=1079.212,414.944,392.921,176.706,31.087,155.495
C03346=1079.219,415.190,392.878,176.710,31.097,155.497
C03347=1079.227,415.436,392.836,176.714,31.107,155.499
C03348=1079.233,415.682,392.794,176.720,31.117,155.501
C03349=1079.240,415.929,392.751,176.724,31.127,155.504
C03350=1079.247,416.174,392.708,176.728,31.137,155.506
C03351=1079.255,416.421,392.665,176.734,31.147,155.508
C03352=1079.262,416.668,392.623,176.738,31.158,155.510
C03353=1079.269,416.914,392.580,176.743,31.168,155.512
C03354=1079.276,417.160,392.537,176.748,31.178,155.515
C03355=1079.283,417.406,392.494,176.753,31.188,155.517
C03356=1079.289,417.652,392.452,176.758,31.199,155.519
C03357=1079.297,417.898,392.408,176.763,31.209,155.522
C03358=1079.304,418.145,392.366,176.767,31.220,155.524
C03359=1079.311,418.391,392.323,176.773,31.230,155.526
C03360=1079.318,418.637,392.280,176.777,31.241,155.529
C03361=1079.325,418.883,392.237,176.782,31.251,155.531
C03362=1079.333,419.129,392.194,176.787,31.262,155.533
C03363=1079.340,419.376,392.151,176.792,31.272,155.535
C03364=1079.347,419.621,392.108,176.797,31.283,155.538
C03365=1079.354,419.868,392.065,176.802,31.293,155.540
C03366=1079.361,420.114,392.022,176.806,31.304,155.543
C03367=1079.369,420.360,391.978,176.812,31.315,155.545
C03368=1079.376,420.607,391.935,176.816,31.325,155.547
C03369=1079.383,420.852,391.892,176.822,31.336,155.550
C03370=1079.390,421.098,391.848,176.826,31.347,155.552
C03371=1079.397,421.345,391.805,176.831,31.358,155.554
C03372=1079.404,421.591,391.762,176.837,31.369,155.557
C03373=1079.412,421.837,391.719,176.841,31.379,155.559
C03374=1079.419,422.083,391.675,176.847,31.390,155.562
C03375=1079.426,422.329,391.632,176.852,31.402,155.564
C03376=1079.433,422.575,391.588,176.857,31.412,155.567
C03377=1079.440,422.821,391.545,176.862,31.423,155.569
C03378=1079.448,423.067,391.501,176.866,31.434,155.571
C03379=1079.455,423.313,391.457,176.872,31.446,155.574
C03380=1079.462,423.559,391.414,176.877,31.457,155.576
C03381=1079.470,423.805,391.370,176.882,31.468,155.579
C03382=1079.476,424.051,391.326,176.887,31.479,155.581
C03383=1079.484,424.297,391.282,176.893,31.491,155.584
C03384=1079.491,424.543,391.239,176.898,31.502,155.586
C03385=1079.498,424.789,391.195,176.902,31.513,155.589
C03386=1079.505,425.035,391.151,176.908,31.524,155.592
C03387=1079.513,425.281,391.106,176.913,31.536,155.594
C03388=1079.521,425.527,391.063,176.919,31.547,155.597
C03389=1079.527,425.784,391.017,176.924,31.559,155.599
C03390=1079.536,426.039,390.971,176.930,31.571,155.602
C03391=1079.543,426.296,390.925,176.935,31.583,155.605
C03392=1079.551,426.553,390.880,176.941,31.595,155.607
C03393=1079.558,426.799,390.835,176.945,31.607,155.610
C03394=1079.565,427.044,390.792,176.951,31.618,155.613
C03395=1079.574,427.290,390.747,176.956,31.630,155.615
C03396=1079.581,427.536,390.702,176.962,31.642,155.618
C03397=1079.588,427.782,390.659,176.967,31.653,155.621
C03398=1079.595,428.028,390.614,176.973,31.665,155.623
C03399=1079.603,428.274,390.570,176.977,31.677,155.626
C03400=1079.610,428.520,390.526,176.983,31.689,155.629
C03401=1079.617,428.766,390.481,176.988,31.701,155.631
C03402=1079.625,429.011,390.437,176.994,31.713,155.634
C03403=1079.633,429.257,390.392,176.999,31.724,155.637
C03404=1079.639,429.503,390.347,177.005,31.737,155.639
C03405=1079.647,429.748,390.303,177.010,31.749,155.642
C03406=1079.655,429.995,390.258,177.016,31.761,155.645
C03407=1079.662,430.241,390.213,177.021,31.773,155.648
C03408=1079.670,430.486,390.169,177.027,31.785,155.650
C03409=1079.677,430.732,390.124,177.032,31.797,155.653
C03410=1079.684,430.978,390.079,177.038,31.810,155.656
C03411=1079.692,431.223,390.035,177.042,31.822,155.659
C03412=1079.700,431.470,389.990,177.048,31.834,155.662
C03413=1079.707,431.716,389.945,177.054,31.846,155.664
C03414=1079.714,431.962,389.900,177.059,31.859,155.667
C03415=1079.723,432.207,389.855,177.066,31.871,155.670
C03416=1079.730,432.453,389.810,177.071,31.884,155.673
C03417=1079.737,432.699,389.765,177.077,31.896,155.676
C03418=1079.745,432.944,389.720,177.083,31.909,155.679
C03419=1079.752,433.190,389.675,177.088,31.922,155.682
C03420=1079.760,433.436,389.629,177.094,31.935,155.685
C03421=1079.767,433.681,389.584,177.099,31.947,155.688
C03422=1079.774,433.927,389.539,177.105,31.960,155.691
C03423=1079.782,434.173,389.494,177.111,31.973,155.693
C03424=1079.789,434.418,389.448,177.116,31.985,155.696
C03425=1079.797,434.664,389.403,177.122,31.999,155.699
C03426=1079.805,434.910,389.357,177.127,32.012,155.702
C03427=1079.812,435.156,389.312,177.134,32.025,155.705
C03428=1079.820,435.401,389.266,177.140,32.037,155.708
C03429=1079.827,435.647,389.221,177.145,32.051,155.711
C03430=1079.835,435.893,389.175,177.151,32.064,155.714
C03431=1079.843,436.138,389.130,177.157,32.077,155.717
C03432=1079.850,436.383,389.084,177.162,32.090,155.721
C03433=1079.858,436.629,389.038,177.169,32.103,155.724
C03434=1079.866,436.874,388.993,177.175,32.116,155.727
C03435=1079.874,437.120,388.947,177.180,32.130,155.730
C03436=1079.882,437.366,388.901,177.186,32.143,155.733
C03437=1079.889,437.611,388.855,177.193,32.156,155.736
C03438=1079.897,437.857,388.810,177.198,32.170,155.739
C03439=1079.905,438.103,388.764,177.204,32.183,155.742
C03440=1079.913,438.348,388.718,177.210,32.197,155.745
C03441=1079.920,438.593,388.671,177.217,32.211,155.749
C03442=1079.927,438.839,388.626,177.222,32.224,155.752
C03443=1079.936,439.085,388.580,177.228,32.238,155.755
C03444=1079.943,439.330,388.534,177.235,32.251,155.758
C03445=1079.951,439.546,388.493,177.240,32.264,155.761
C03446=1079.957,439.763,388.452,177.245,32.276,155.764
C03447=1079.964,439.979,388.412,177.251,32.288,155.767
C03448=1079.971,440.195,388.370,177.256,32.300,155.770
C03449=1079.978,440.412,388.330,177.262,32.312,155.772
C03450=1079.985,440.628,388.289,177.267,32.325,155.775
C03451=1079.992,440.844,388.248,177.272,32.337,155.778
C03452=1079.998,441.060,388.207,177.278,32.349,155.781
C03453=1080.007,441.306,388.160,177.284,32.364,155.784
C03454=1080.015,441.551,388.114,177.291,32.378,155.788
C03455=1080.022,441.797,388.068,177.297,32.392,155.791
C03456=1080.030,442.042,388.021,177.303,32.406,155.795
C03457=1080.038,442.288,387.974,177.309,32.421,155.798
C03458=1080.046,442.533,387.927,177.316,32.435,155.801
C03459=1080.054,442.779,387.880,177.322,32.450,155.805
C03460=1080.062,443.023,387.834,177.329,32.464,155.808
C03461=1080.069,443.269,387.786,177.335,32.479,155.812
C03462=1080.077,443.514,387.740,177.341,32.493,155.815
C03463=1080.085,443.760,387.693,177.347,32.507,155.818
C03464=1080.094,444.005,387.646,177.354,32.522,155.822
C03465=1080.101,444.250,387.599,177.360,32.537,155.825
C03466=1080.110,444.496,387.552,177.367,32.552,155.829
C03467=1080.117,444.742,387.505,177.374,32.567,155.833
C03468=1080.125,444.987,387.459,177.380,32.582,155.836
C03469=1080.133,445.232,387.411,177.387,32.597,155.840
C03470=1080.141,445.478,387.363,177.394,32.611,155.843
C03471=1080.149,445.722,387.316,177.400,32.627,155.847
C03472=1080.157,445.968,387.269,177.407,32.642,155.850
C03473=1080.165,446.213,387.221,177.413,32.657,155.854
C03474=1080.174,446.458,387.174,177.419,32.672,155.858
C03475=1080.181,446.703,387.126,177.425,32.687,155.861
C03476=1080.189,446.949,387.079,177.431,32.702,155.865
C03477=1080.198,447.194,387.032,177.436,32.718,155.869
C03478=1080.206,447.439,386.984,177.441,32.732,155.872
C03479=1080.214,447.685,386.936,177.446,32.747,155.876
C03480=1080.222,447.930,386.888,177.451,32.762,155.880
C03481=1080.231,448.175,386.841,177.455,32.778,155.883
C03482=1080.238,448.420,386.794,177.459,32.792,155.887
C03483=1080.246,448.665,386.746,177.463,32.808,155.891
C03484=1080.254,448.910,386.698,177.467,32.822,155.895
C03485=1080.263,449.155,386.650,177.470,32.837,155.898
C03486=1080.273,449.400,386.604,177.473,32.852,155.902
C03487=1080.285,449.646,386.558,177.477,32.865,155.905
C03488=1080.298,449.891,386.513,177.481,32.878,155.908
C03489=1079.933,449.885,386.290,177.455,33.045,155.953
C03490=1079.920,449.640,386.335,177.451,33.032,155.950
C03491=1079.908,449.394,386.381,177.447,33.019,155.946
C03492=1079.897,449.149,386.427,177.444,33.005,155.943
C03493=1079.889,448.905,386.475,177.440,32.990,155.939
C03494=1079.881,448.660,386.523,177.437,32.975,155.935
C03495=1079.873,448.414,386.571,177.432,32.960,155.932
C03496=1079.864,448.169,386.618,177.428,32.945,155.928
C03497=1079.856,447.924,386.666,177.423,32.930,155.924
C03498=1079.848,447.679,386.714,177.418,32.915,155.920
C03499=1079.840,447.434,386.762,177.414,32.900,155.917
C03500=1079.831,447.188,386.809,177.408,32.885,155.913
C03501=1079.823,446.943,386.857,177.402,32.869,155.909
C03502=1079.815,446.698,386.905,177.396,32.854,155.906
C03503=1079.808,446.452,386.952,177.390,32.839,155.902
C03504=1079.799,446.208,386.999,177.384,32.824,155.898
C03505=1079.791,445.962,387.047,177.378,32.809,155.895
C03506=1079.783,445.717,387.095,177.371,32.794,155.891
C03507=1079.775,445.472,387.142,177.365,32.779,155.888
C03508=1079.767,445.227,387.189,177.358,32.764,155.884
C03509=1079.759,444.981,387.236,177.351,32.749,155.880
C03510=1079.750,444.736,387.284,177.345,32.734,155.877
C03511=1079.743,444.491,387.331,177.338,32.719,155.873
C03512=1079.735,444.245,387.378,177.331,32.704,155.870
C03513=1079.726,444.000,387.426,177.325,32.690,155.866
C03514=1079.719,443.755,387.472,177.318,32.675,155.863
C03515=1079.711,443.509,387.519,177.312,32.660,155.859
C03516=1079.702,443.264,387.566,177.305,32.646,155.856
C03517=1079.695,443.019,387.613,177.299,32.631,155.852
C03518=1079.686,442.773,387.660,177.292,32.617,155.849
C03519=1079.679,442.528,387.707,177.286,32.603,155.846
C03520=1079.671,442.283,387.753,177.279,32.588,155.842
C03521=1079.663,442.037,387.800,177.273,32.574,155.839
C03522=1079.655,441.792,387.847,177.266,32.559,155.835
C03523=1079.647,441.546,387.894,177.260,32.545,155.832
C03524=1079.639,441.301,387.940,177.254,32.531,155.829
C03525=1079.632,441.056,387.986,177.248,32.517,155.825
C03526=1079.624,440.848,388.026,177.242,32.505,155.822
C03527=1079.618,440.639,388.066,177.237,32.493,155.820
C03528=1079.612,440.431,388.105,177.231,32.481,155.817
C03529=1079.604,440.223,388.145,177.226,32.469,155.814
C03530=1079.598,440.015,388.183,177.221,32.457,155.811
C03531=1079.592,439.807,388.223,177.215,32.446,155.809
C03532=1079.585,439.599,388.262,177.211,32.434,155.806
C03533=1079.578,439.390,388.302,177.205,32.422,155.803
C03534=1079.571,439.145,388.347,177.199,32.409,155.800
C03535=1079.562,438.900,388.394,177.193,32.395,155.797
C03536=1079.554,438.654,388.440,177.186,32.381,155.793
C03537=1079.547,438.409,388.485,177.180,32.368,155.790
C03538=1079.539,438.162,388.532,177.175,32.354,155.787
C03539=1079.531,437.917,388.578,177.169,32.341,155.784
C03540=1079.524,437.672,388.624,177.162,32.327,155.781
C03541=1079.515,437.426,388.670,177.156,32.314,155.778
C03542=1079.508,437.180,388.716,177.150,32.300,155.774
C03543=1079.500,436.935,388.761,177.145,32.287,155.771
C03544=1079.492,436.690,388.807,177.138,32.274,155.768
C03545=1079.484,436.443,388.853,177.132,32.261,155.765
C03546=1079.477,436.198,388.899,177.126,32.248,155.762
C03547=1079.469,435.953,388.944,177.121,32.234,155.759
C03548=1079.461,435.707,388.990,177.115,32.221,155.756
C03549=1079.454,435.462,389.036,177.108,32.208,155.753
C03550=1079.446,435.216,389.081,177.102,32.195,155.750
C03551=1079.439,434.970,389.126,177.097,32.182,155.747
C03552=1079.430,434.724,389.172,177.091,32.169,155.744
C03553=1079.423,434.479,389.218,177.085,32.156,155.741
C03554=1079.415,434.233,389.263,177.080,32.143,155.738
C03555=1079.408,433.987,389.308,177.074,32.131,155.735
C03556=1079.400,433.742,389.354,177.068,32.118,155.732
C03557=1079.393,433.496,389.399,177.062,32.105,155.729
C03558=1079.385,433.250,389.445,177.056,32.092,155.726
C03559=1079.378,433.004,389.490,177.050,32.080,155.723
C03560=1079.370,432.759,389.535,177.044,32.067,155.721
C03561=1079.364,432.513,389.580,177.039,32.054,155.718
C03562=1079.356,432.268,389.625,177.033,32.042,155.715
C03563=1079.349,432.022,389.670,177.027,32.029,155.712
C03564=1079.340,431.776,389.715,177.022,32.017,155.709
C03565=1079.333,431.531,389.760,177.016,32.004,155.706
C03566=1079.326,431.285,389.805,177.010,31.992,155.703
C03567=1079.318,431.039,389.850,177.005,31.980,155.701
C03568=1079.310,430.793,389.895,176.999,31.968,155.698
C03569=1079.303,430.547,389.939,176.994,31.955,155.695
C03570=1079.295,430.301,389.984,176.988,31.943,155.692
C03571=1079.287,430.055,390.029,176.983,31.931,155.689
C03572=1079.280,429.809,390.074,176.978,31.919,155.687
C03573=1079.273,429.564,390.118,176.972,31.907,155.684
C03574=1079.265,429.318,390.163,176.967,31.895,155.681
C03575=1079.258,429.072,390.208,176.961,31.883,155.678
C03576=1079.251,428.826,390.252,176.955,31.871,155.676
C03577=1079.243,428.581,390.296,176.950,31.859,155.673
C03578=1079.236,428.335,390.341,176.944,31.847,155.670
C03579=1079.228,428.089,390.386,176.939,31.835,155.668
C03580=1079.221,427.842,390.430,176.934,31.824,155.665
C03581=1079.213,427.596,390.475,176.928,31.812,155.662
C03582=1079.206,427.351,390.519,176.923,31.800,155.660
C03583=1079.198,427.105,390.562,176.917,31.788,155.657
C03584=1079.191,426.859,390.607,176.912,31.777,155.654
C03585=1079.183,426.614,390.651,176.907,31.765,155.652
C03586=1079.176,426.356,390.697,176.901,31.753,155.649
C03587=1079.169,426.098,390.744,176.895,31.741,155.646
C03588=1079.161,425.840,390.790,176.890,31.729,155.644
C03589=1079.153,425.583,390.836,176.884,31.717,155.641
C03590=1079.145,425.336,390.880,176.879,31.706,155.638
C03591=1079.138,425.090,390.924,176.874,31.694,155.636
C03592=1079.130,424.845,390.968,176.868,31.683,155.633
C03593=1079.123,424.598,391.012,176.863,31.671,155.631
C03594=1079.116,424.352,391.056,176.858,31.660,155.628
C03595=1079.108,424.106,391.099,176.853,31.649,155.626
C03596=1079.101,423.861,391.143,176.847,31.638,155.623
C03597=1079.094,423.614,391.188,176.843,31.627,155.621
C03598=1079.087,423.369,391.231,176.837,31.615,155.618
C03599=1079.079,423.122,391.274,176.832,31.604,155.616
C03600=1079.073,422.876,391.318,176.827,31.593,155.613
C03601=1079.065,422.630,391.362,176.822,31.582,155.611
C03602=1079.058,422.384,391.405,176.816,31.571,155.608
C03603=1079.051,422.138,391.449,176.812,31.560,155.606
C03604=1079.044,421.892,391.493,176.806,31.549,155.603
C03605=1079.036,421.646,391.536,176.802,31.538,155.601
C03606=1079.029,421.400,391.580,176.796,31.527,155.598
C03607=1079.021,421.154,391.623,176.791,31.517,155.596
C03608=1079.014,420.908,391.666,176.786,31.506,155.594
C03609=1079.008,420.661,391.710,176.781,31.495,155.591
C03610=1079.000,420.416,391.753,176.776,31.484,155.589
C03611=1078.993,420.169,391.796,176.771,31.473,155.586
C03612=1078.985,419.924,391.840,176.767,31.463,155.584
C03613=1078.979,419.677,391.882,176.761,31.452,155.582
C03614=1078.971,419.431,391.926,176.757,31.442,155.579
C03615=1078.964,419.185,391.968,176.751,31.431,155.577
C03616=1078.957,418.939,392.012,176.746,31.420,155.575
C03617=1078.949,418.693,392.055,176.741,31.410,155.572
C03618=1078.942,418.446,392.098,176.737,31.400,155.570
C03619=1078.935,418.201,392.141,176.731,31.389,155.568
C03620=1078.928,417.954,392.184,176.727,31.379,155.565
C03621=1078.921,417.707,392.226,176.721,31.368,155.563
C03622=1078.914,417.462,392.270,176.717,31.358,155.561
C03623=1078.907,417.215,392.312,176.712,31.347,155.559
C03624=1078.900,416.969,392.355,176.707,31.337,155.556
C03625=1078.893,416.723,392.398,176.702,31.327,155.554
C03626=1078.885,416.476,392.441,176.697,31.317,155.552
C03627=1078.878,416.230,392.484,176.693,31.307,155.550
C03628=1078.871,415.985,392.527,176.687,31.296,155.547
C03629=1078.864,415.738,392.569,176.683,31.286,155.545
C03630=1078.858,415.492,392.612,176.678,31.276,155.543
C03631=1078.850,415.246,392.654,176.673,31.266,155.541
C03632=1078.842,414.999,392.697,176.669,31.256,155.538
C03633=1078.836,414.753,392.739,176.663,31.246,155.536
C03634=1078.829,414.506,392.782,176.659,31.236,155.534
C03635=1078.821,414.260,392.824,176.654,31.226,155.532
C03636=1078.814,414.014,392.866,176.649,31.216,155.530
C03637=1078.807,413.768,392.909,176.645,31.206,155.528
C03638=1078.800,413.524,392.950,176.640,31.197,155.526
C03639=1078.793,413.280,392.992,176.635,31.187,155.523
C03640=1078.786,413.038,393.034,176.630,31.177,155.521
